REGION Network 65: [Ax] Movimento PTRK da Pos1 Ribalta + Tempo Assestamento ==a==> Pos2 Ribalta
   RUNG wire#powerrail
      "PTrk_Presence"(Item := "PTrk".A0301.P["PTRK_A0301_Ribalta_Pos1"])
      "PTrk_Absence"(Item := "PTrk".A0301.P["PTRK_A0301_Ribalta_Pos2"])
      I_Contact( #Ctrl.TRK.Ribaltatore.MoveToPos1 )
      Contact( #CIn.Ribaltatore.Solleva_Rib.Work )
      Contact( #CIn.Ribaltatore.Sts_Ribaltatore.Pos1_Reached )
      { S7_Templates := "time_type := Time" } #TON.Delay_Pos1Ribalta.TON(pt := "PPrf_MAIN".ON_WORK.A0301_A0302.Ribaltatore.Pos_1_Delay, et =>)
      Contact( #TON.Delay_Pos1Ribalta.Q )
      wire#w1
      I_Contact( #CIn.Ribaltatore.Sts_Ribaltatore.Pos2_Reached )
      wire#w2
      Coil( #Ctrl.TRK.Ribaltatore.MoveToPos2 )
   END_RUNG
   RUNG wire#powerrail
      "PTrk_Presence"(Item := "PTrk".A0301.P["PTRK_A0301_Ribalta_Pos2"])
      I_Contact( #Ctrl.TRK.Ribaltatore.MoveToPos1 )
      I_Contact( #Ctrl.TRK.Ribaltatore.MoveToPos3 )
   END_RUNG wire#w1
   RUNG wire#powerrail
      Contact( #Ctrl.TRK.Ribaltatore.MoveToPos2 )
      I_Contact( #CIn.Ribaltatore.Sts_Ribaltatore.Pos2_Reached )
   END_RUNG wire#w2
   RUNG wire#powerrail
      I_Contact( #Ctrl.TRK.Ribaltatore.MoveToPos2 )
      Contact( #CIn.Ribaltatore.Sts_Ribaltatore.Pos2_Reached )
      "PTrk_Presence"(Item := "PTrk".A0301.P["PTRK_A0301_Ribalta_Pos1"])
      "PTrk_Absence"(Item := "PTrk".A0301.P["PTRK_A0301_Ribalta_Pos2"])
      Move(in := "PTrk".A0301.P["PTRK_A0301_Ribalta_Pos1"], out1 => "PTrk".A0301.P["PTRK_A0301_Ribalta_Pos2"])
      "PTrk_Presence"(Item := "PTrk".A0301.P["PTRK_A0301_Ribalta_Pos2"])
      Move(in := "PTrk".Empty, out1 => "PTrk".A0301.P["PTRK_A0301_Ribalta_Pos1"])
   END_RUNG
   // the same network as SCL:
   "PTrk_Presence"(Item := "PTrk".A0301.P["PTRK_A0301_Ribalta_Pos1"], ENO => #_w1);
   "PTrk_Absence"(EN := #_w1, Item := "PTrk".A0301.P["PTRK_A0301_Ribalta_Pos2"], ENO => #_w2);
   #TON.Delay_Pos1Ribalta.TON(IN := #_w2 AND NOT #Ctrl.TRK.Ribaltatore.MoveToPos1 AND #CIn.Ribaltatore.Solleva_Rib.Work AND #CIn.Ribaltatore.Sts_Ribaltatore.Pos1_Reached,
                           PT := "PPrf_MAIN".ON_WORK.A0301_A0302.Ribaltatore.Pos_1_Delay);
   "PTrk_Presence"(Item := "PTrk".A0301.P["PTRK_A0301_Ribalta_Pos2"], ENO => #_w3);
   #Ctrl.TRK.Ribaltatore.MoveToPos2 := (((#TON.Delay_Pos1Ribalta.Q AND #TON.Delay_Pos1Ribalta.Q) OR (#_w3 AND NOT #Ctrl.TRK.Ribaltatore.MoveToPos1 AND NOT #Ctrl.TRK.Ribaltatore.MoveToPos3)) AND NOT #CIn.Ribaltatore.Sts_Ribaltatore.Pos2_Reached) OR (#Ctrl.TRK.Ribaltatore.MoveToPos2 AND NOT #CIn.Ribaltatore.Sts_Ribaltatore.Pos2_Reached);
   "PTrk_Presence"(EN := NOT #Ctrl.TRK.Ribaltatore.MoveToPos2 AND #CIn.Ribaltatore.Sts_Ribaltatore.Pos2_Reached,
                   Item := "PTrk".A0301.P["PTRK_A0301_Ribalta_Pos1"],
                   ENO => #_w4);
   "PTrk_Absence"(EN := #_w4, Item := "PTrk".A0301.P["PTRK_A0301_Ribalta_Pos2"], ENO => #_w5);
   IF #_w5 THEN
       "PTrk".A0301.P["PTRK_A0301_Ribalta_Pos2"] := "PTrk".A0301.P["PTRK_A0301_Ribalta_Pos1"];
   END_IF;
   "PTrk_Presence"(EN := #_w5, Item := "PTrk".A0301.P["PTRK_A0301_Ribalta_Pos2"], ENO => #_w6);
   IF #_w6 THEN "PTrk".A0301.P["PTRK_A0301_Ribalta_Pos1"] := "PTrk".Empty; END_IF;
END_REGION

REGION Network 66: [Ax] Movimento PTRK da Pos2 Ribalta ==a==> Pos3 Ribalta
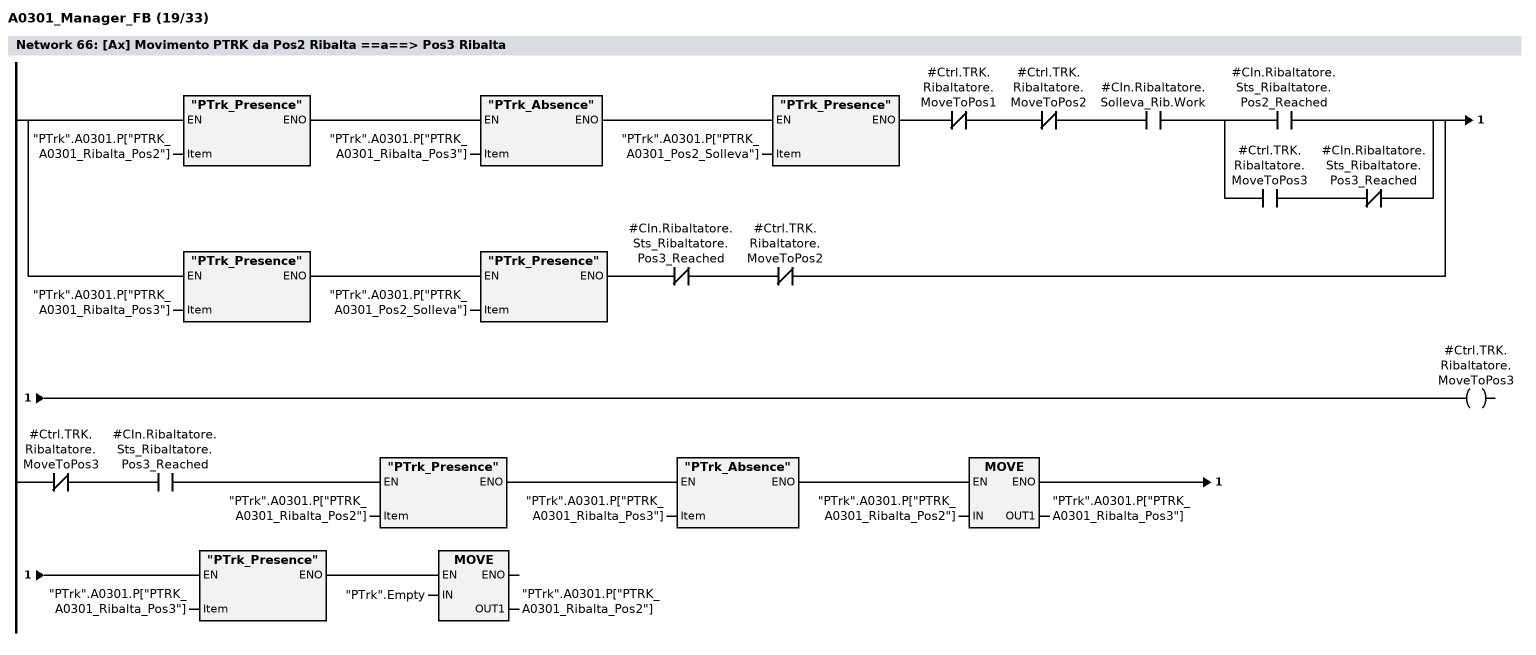
   RUNG wire#powerrail
      "PTrk_Presence"(Item := "PTrk".A0301.P["PTRK_A0301_Ribalta_Pos2"])
      "PTrk_Absence"(Item := "PTrk".A0301.P["PTRK_A0301_Ribalta_Pos3"])
      "PTrk_Presence"(Item := "PTrk".A0301.P["PTRK_A0301_Pos2_Solleva"])
      I_Contact( #Ctrl.TRK.Ribaltatore.MoveToPos1 )
      I_Contact( #Ctrl.TRK.Ribaltatore.MoveToPos2 )
      Contact( #CIn.Ribaltatore.Solleva_Rib.Work )
      wire#w1
      Contact( #CIn.Ribaltatore.Sts_Ribaltatore.Pos2_Reached )
      wire#w2
      Coil( #Ctrl.TRK.Ribaltatore.MoveToPos3 )
   END_RUNG
   RUNG wire#w1
      Contact( #Ctrl.TRK.Ribaltatore.MoveToPos3 )
      I_Contact( #CIn.Ribaltatore.Sts_Ribaltatore.Pos3_Reached )
   END_RUNG wire#w2
   RUNG wire#powerrail
      "PTrk_Presence"(Item := "PTrk".A0301.P["PTRK_A0301_Ribalta_Pos3"])
      "PTrk_Presence"(Item := "PTrk".A0301.P["PTRK_A0301_Pos2_Solleva"])
      I_Contact( #CIn.Ribaltatore.Sts_Ribaltatore.Pos3_Reached )
      I_Contact( #Ctrl.TRK.Ribaltatore.MoveToPos2 )
   END_RUNG wire#w2
   RUNG wire#powerrail
      I_Contact( #Ctrl.TRK.Ribaltatore.MoveToPos3 )
      Contact( #CIn.Ribaltatore.Sts_Ribaltatore.Pos3_Reached )
      "PTrk_Presence"(Item := "PTrk".A0301.P["PTRK_A0301_Ribalta_Pos2"])
      "PTrk_Absence"(Item := "PTrk".A0301.P["PTRK_A0301_Ribalta_Pos3"])
      Move(in := "PTrk".A0301.P["PTRK_A0301_Ribalta_Pos2"], out1 => "PTrk".A0301.P["PTRK_A0301_Ribalta_Pos3"])
      "PTrk_Presence"(Item := "PTrk".A0301.P["PTRK_A0301_Ribalta_Pos3"])
      Move(in := "PTrk".Empty, out1 => "PTrk".A0301.P["PTRK_A0301_Ribalta_Pos2"])
   END_RUNG
   // the same network as SCL:
   "PTrk_Presence"(Item := "PTrk".A0301.P["PTRK_A0301_Ribalta_Pos2"], ENO => #_w1);
   "PTrk_Absence"(EN := #_w1, Item := "PTrk".A0301.P["PTRK_A0301_Ribalta_Pos3"], ENO => #_w2);
   "PTrk_Presence"(EN := #_w2, Item := "PTrk".A0301.P["PTRK_A0301_Pos2_Solleva"], ENO => #_w3);
   "PTrk_Presence"(Item := "PTrk".A0301.P["PTRK_A0301_Ribalta_Pos3"], ENO => #_w4);
   "PTrk_Presence"(EN := #_w4, Item := "PTrk".A0301.P["PTRK_A0301_Pos2_Solleva"], ENO => #_w5);
   #Ctrl.TRK.Ribaltatore.MoveToPos3 := (#_w3 AND NOT #Ctrl.TRK.Ribaltatore.MoveToPos1 AND NOT #Ctrl.TRK.Ribaltatore.MoveToPos2 AND #CIn.Ribaltatore.Solleva_Rib.Work AND (#CIn.Ribaltatore.Sts_Ribaltatore.Pos2_Reached OR (#Ctrl.TRK.Ribaltatore.MoveToPos3 AND NOT #CIn.Ribaltatore.Sts_Ribaltatore.Pos3_Reached))) OR (#_w5 AND NOT #CIn.Ribaltatore.Sts_Ribaltatore.Pos3_Reached AND NOT #Ctrl.TRK.Ribaltatore.MoveToPos2);
   "PTrk_Presence"(EN := NOT #Ctrl.TRK.Ribaltatore.MoveToPos3 AND #CIn.Ribaltatore.Sts_Ribaltatore.Pos3_Reached,
                   Item := "PTrk".A0301.P["PTRK_A0301_Ribalta_Pos2"],
                   ENO => #_w6);
   "PTrk_Absence"(EN := #_w6, Item := "PTrk".A0301.P["PTRK_A0301_Ribalta_Pos3"], ENO => #_w7);
   IF #_w7 THEN
       "PTrk".A0301.P["PTRK_A0301_Ribalta_Pos3"] := "PTrk".A0301.P["PTRK_A0301_Ribalta_Pos2"];
   END_IF;
   "PTrk_Presence"(EN := #_w7, Item := "PTrk".A0301.P["PTRK_A0301_Ribalta_Pos3"], ENO => #_w8);
   IF #_w8 THEN "PTrk".A0301.P["PTRK_A0301_Ribalta_Pos2"] := "PTrk".Empty; END_IF;
END_REGION

REGION Network 67: <+>
END_REGION

REGION Network 68: << GESTIONE MOVIMENTO RIBALTATORE / SOLLEVA RIBALTATORE >>
END_REGION

REGION Network 69: [Ax] Ribaltatore - COut Manager
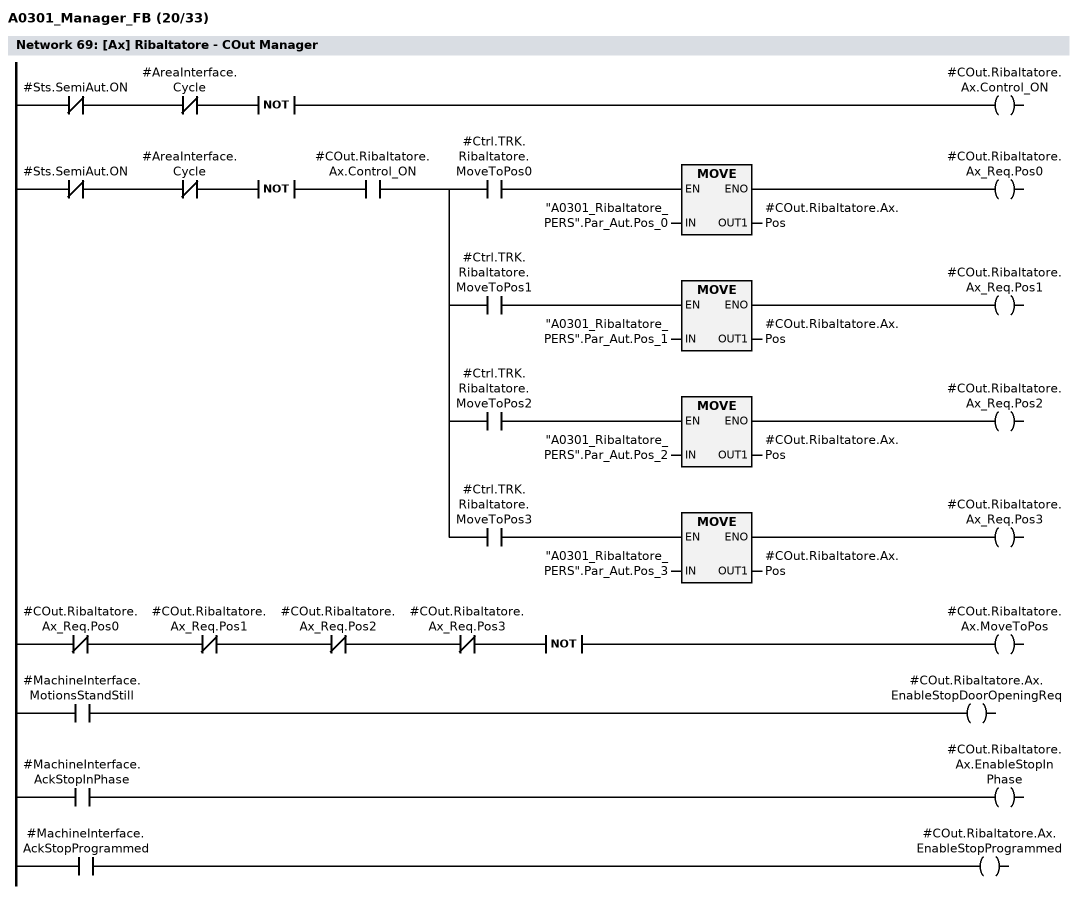
   RUNG wire#powerrail
      I_Contact( #Sts.SemiAut.ON )
      I_Contact( #AreaInterface.Cycle )
      Not()
      Coil( #COut.Ribaltatore.Ax.Control_ON )
   END_RUNG
   RUNG wire#powerrail
      I_Contact( #Sts.SemiAut.ON )
      I_Contact( #AreaInterface.Cycle )
      Not()
      Contact( #COut.Ribaltatore.Ax.Control_ON )
      wire#w1
      Contact( #Ctrl.TRK.Ribaltatore.MoveToPos0 )
      Move(in := "A0301_Ribaltatore_PERS".Par_Aut.Pos_0, out1 => #COut.Ribaltatore.Ax.Pos)
      Coil( #COut.Ribaltatore.Ax_Req.Pos0 )
   END_RUNG
   RUNG wire#w1
      Contact( #Ctrl.TRK.Ribaltatore.MoveToPos1 )
      Move(in := "A0301_Ribaltatore_PERS".Par_Aut.Pos_1, out1 => #COut.Ribaltatore.Ax.Pos)
      Coil( #COut.Ribaltatore.Ax_Req.Pos1 )
   END_RUNG
   RUNG wire#w1
      Contact( #Ctrl.TRK.Ribaltatore.MoveToPos2 )
      Move(in := "A0301_Ribaltatore_PERS".Par_Aut.Pos_2, out1 => #COut.Ribaltatore.Ax.Pos)
      Coil( #COut.Ribaltatore.Ax_Req.Pos2 )
   END_RUNG
   RUNG wire#w1
      Contact( #Ctrl.TRK.Ribaltatore.MoveToPos3 )
      Move(in := "A0301_Ribaltatore_PERS".Par_Aut.Pos_3, out1 => #COut.Ribaltatore.Ax.Pos)
      Coil( #COut.Ribaltatore.Ax_Req.Pos3 )
   END_RUNG
   RUNG wire#powerrail
      I_Contact( #COut.Ribaltatore.Ax_Req.Pos0 )
      I_Contact( #COut.Ribaltatore.Ax_Req.Pos1 )
      I_Contact( #COut.Ribaltatore.Ax_Req.Pos2 )
      I_Contact( #COut.Ribaltatore.Ax_Req.Pos3 )
      Not()
      Coil( #COut.Ribaltatore.Ax.MoveToPos )
   END_RUNG
   RUNG wire#powerrail
      Contact( #MachineInterface.MotionsStandStill )
      Coil( #COut.Ribaltatore.Ax.EnableStopDoorOpeningReq )
   END_RUNG
   RUNG wire#powerrail
      Contact( #MachineInterface.AckStopInPhase )
      Coil( #COut.Ribaltatore.Ax.EnableStopInPhase )
   END_RUNG
   RUNG wire#powerrail
      Contact( #MachineInterface.AckStopProgrammed )
      Coil( #COut.Ribaltatore.Ax.EnableStopProgrammed )
   END_RUNG
   // the same network as SCL:
   #COut.Ribaltatore.Ax.Control_ON := NOT (NOT #Sts.SemiAut.ON AND NOT #AreaInterface.Cycle);
   #_w1 := NOT (NOT #Sts.SemiAut.ON AND NOT #AreaInterface.Cycle) AND #COut.Ribaltatore.Ax.Control_ON;
   #_w2 := #_w1 AND #Ctrl.TRK.Ribaltatore.MoveToPos0;
   IF #_w2 THEN #COut.Ribaltatore.Ax.Pos := "A0301_Ribaltatore_PERS".Par_Aut.Pos_0; END_IF;
   #COut.Ribaltatore.Ax_Req.Pos0 := #_w2;
   #_w3 := #_w1 AND #Ctrl.TRK.Ribaltatore.MoveToPos1;
   IF #_w3 THEN #COut.Ribaltatore.Ax.Pos := "A0301_Ribaltatore_PERS".Par_Aut.Pos_1; END_IF;
   #COut.Ribaltatore.Ax_Req.Pos1 := #_w3;
   #_w4 := #_w1 AND #Ctrl.TRK.Ribaltatore.MoveToPos2;
   IF #_w4 THEN #COut.Ribaltatore.Ax.Pos := "A0301_Ribaltatore_PERS".Par_Aut.Pos_2; END_IF;
   #COut.Ribaltatore.Ax_Req.Pos2 := #_w4;
   #_w5 := #_w1 AND #Ctrl.TRK.Ribaltatore.MoveToPos3;
   IF #_w5 THEN #COut.Ribaltatore.Ax.Pos := "A0301_Ribaltatore_PERS".Par_Aut.Pos_3; END_IF;
   #COut.Ribaltatore.Ax_Req.Pos3 := #_w5;
   #COut.Ribaltatore.Ax.MoveToPos := NOT (NOT #COut.Ribaltatore.Ax_Req.Pos0 AND NOT #COut.Ribaltatore.Ax_Req.Pos1 AND NOT #COut.Ribaltatore.Ax_Req.Pos2 AND NOT #COut.Ribaltatore.Ax_Req.Pos3);
   #COut.Ribaltatore.Ax.EnableStopDoorOpeningReq := #MachineInterface.MotionsStandStill;
   #COut.Ribaltatore.Ax.EnableStopInPhase := #MachineInterface.AckStopInPhase;
   #COut.Ribaltatore.Ax.EnableStopProgrammed := #MachineInterface.AckStopProgrammed;
END_REGION

REGION Network 70: [Ax] Ribaltatore - RIFERIMENTI Velocità
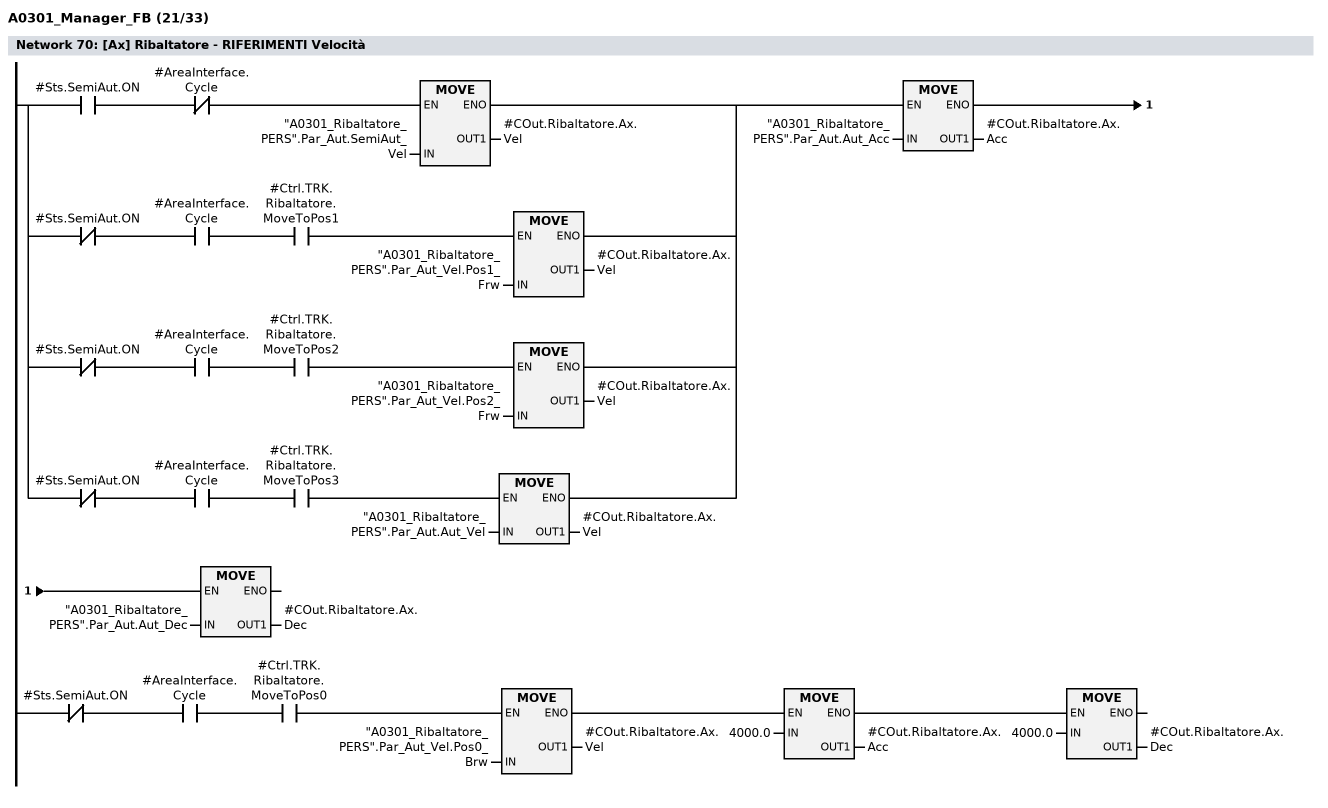
   RUNG wire#powerrail
      Contact( #Sts.SemiAut.ON )
      I_Contact( #AreaInterface.Cycle )
      Move(in := "A0301_Ribaltatore_PERS".Par_Aut.SemiAut_Vel, out1 => #COut.Ribaltatore.Ax.Vel)
      wire#w1
      Move(in := "A0301_Ribaltatore_PERS".Par_Aut.Aut_Acc, out1 => #COut.Ribaltatore.Ax.Acc)
      Move(in := "A0301_Ribaltatore_PERS".Par_Aut.Aut_Dec, out1 => #COut.Ribaltatore.Ax.Dec)
   END_RUNG
   RUNG wire#powerrail
      I_Contact( #Sts.SemiAut.ON )
      Contact( #AreaInterface.Cycle )
      Contact( #Ctrl.TRK.Ribaltatore.MoveToPos1 )
      Move(in := "A0301_Ribaltatore_PERS".Par_Aut_Vel.Pos1_Frw, out1 => #COut.Ribaltatore.Ax.Vel)
   END_RUNG wire#w1
   RUNG wire#powerrail
      I_Contact( #Sts.SemiAut.ON )
      Contact( #AreaInterface.Cycle )
      Contact( #Ctrl.TRK.Ribaltatore.MoveToPos2 )
      Move(in := "A0301_Ribaltatore_PERS".Par_Aut_Vel.Pos2_Frw, out1 => #COut.Ribaltatore.Ax.Vel)
   END_RUNG wire#w1
   RUNG wire#powerrail
      I_Contact( #Sts.SemiAut.ON )
      Contact( #AreaInterface.Cycle )
      Contact( #Ctrl.TRK.Ribaltatore.MoveToPos3 )
      Move(in := "A0301_Ribaltatore_PERS".Par_Aut.Aut_Vel, out1 => #COut.Ribaltatore.Ax.Vel)
   END_RUNG wire#w1
   RUNG wire#powerrail
      I_Contact( #Sts.SemiAut.ON )
      Contact( #AreaInterface.Cycle )
      Contact( #Ctrl.TRK.Ribaltatore.MoveToPos0 )
      Move(in := "A0301_Ribaltatore_PERS".Par_Aut_Vel.Pos0_Brw, out1 => #COut.Ribaltatore.Ax.Vel)
      Move(in := 4000.0, out1 => #COut.Ribaltatore.Ax.Acc)
      Move(in := 4000.0, out1 => #COut.Ribaltatore.Ax.Dec)
   END_RUNG
   // the same network as SCL:
   #_w1 := #Sts.SemiAut.ON AND NOT #AreaInterface.Cycle;
   IF #_w1 THEN #COut.Ribaltatore.Ax.Vel := "A0301_Ribaltatore_PERS".Par_Aut.SemiAut_Vel; END_IF;
   #_w2 := NOT #Sts.SemiAut.ON AND #AreaInterface.Cycle AND #Ctrl.TRK.Ribaltatore.MoveToPos1;
   IF #_w2 THEN #COut.Ribaltatore.Ax.Vel := "A0301_Ribaltatore_PERS".Par_Aut_Vel.Pos1_Frw; END_IF;
   #_w3 := NOT #Sts.SemiAut.ON AND #AreaInterface.Cycle AND #Ctrl.TRK.Ribaltatore.MoveToPos2;
   IF #_w3 THEN #COut.Ribaltatore.Ax.Vel := "A0301_Ribaltatore_PERS".Par_Aut_Vel.Pos2_Frw; END_IF;
   #_w4 := NOT #Sts.SemiAut.ON AND #AreaInterface.Cycle AND #Ctrl.TRK.Ribaltatore.MoveToPos3;
   IF #_w4 THEN #COut.Ribaltatore.Ax.Vel := "A0301_Ribaltatore_PERS".Par_Aut.Aut_Vel; END_IF;
   IF #_w1 OR #_w2 OR #_w3 OR #_w4 THEN
       #COut.Ribaltatore.Ax.Acc := "A0301_Ribaltatore_PERS".Par_Aut.Aut_Acc;
       #COut.Ribaltatore.Ax.Dec := "A0301_Ribaltatore_PERS".Par_Aut.Aut_Dec;
   END_IF;
   IF NOT #Sts.SemiAut.ON AND #AreaInterface.Cycle AND #Ctrl.TRK.Ribaltatore.MoveToPos0 THEN
       #COut.Ribaltatore.Ax.Vel := "A0301_Ribaltatore_PERS".Par_Aut_Vel.Pos0_Brw;
       #COut.Ribaltatore.Ax.Acc := 4000.0;
       #COut.Ribaltatore.Ax.Dec := 4000.0;
   END_IF;
END_REGION

REGION Network 71: P [Solleva] Ribaltatore - COut Manager
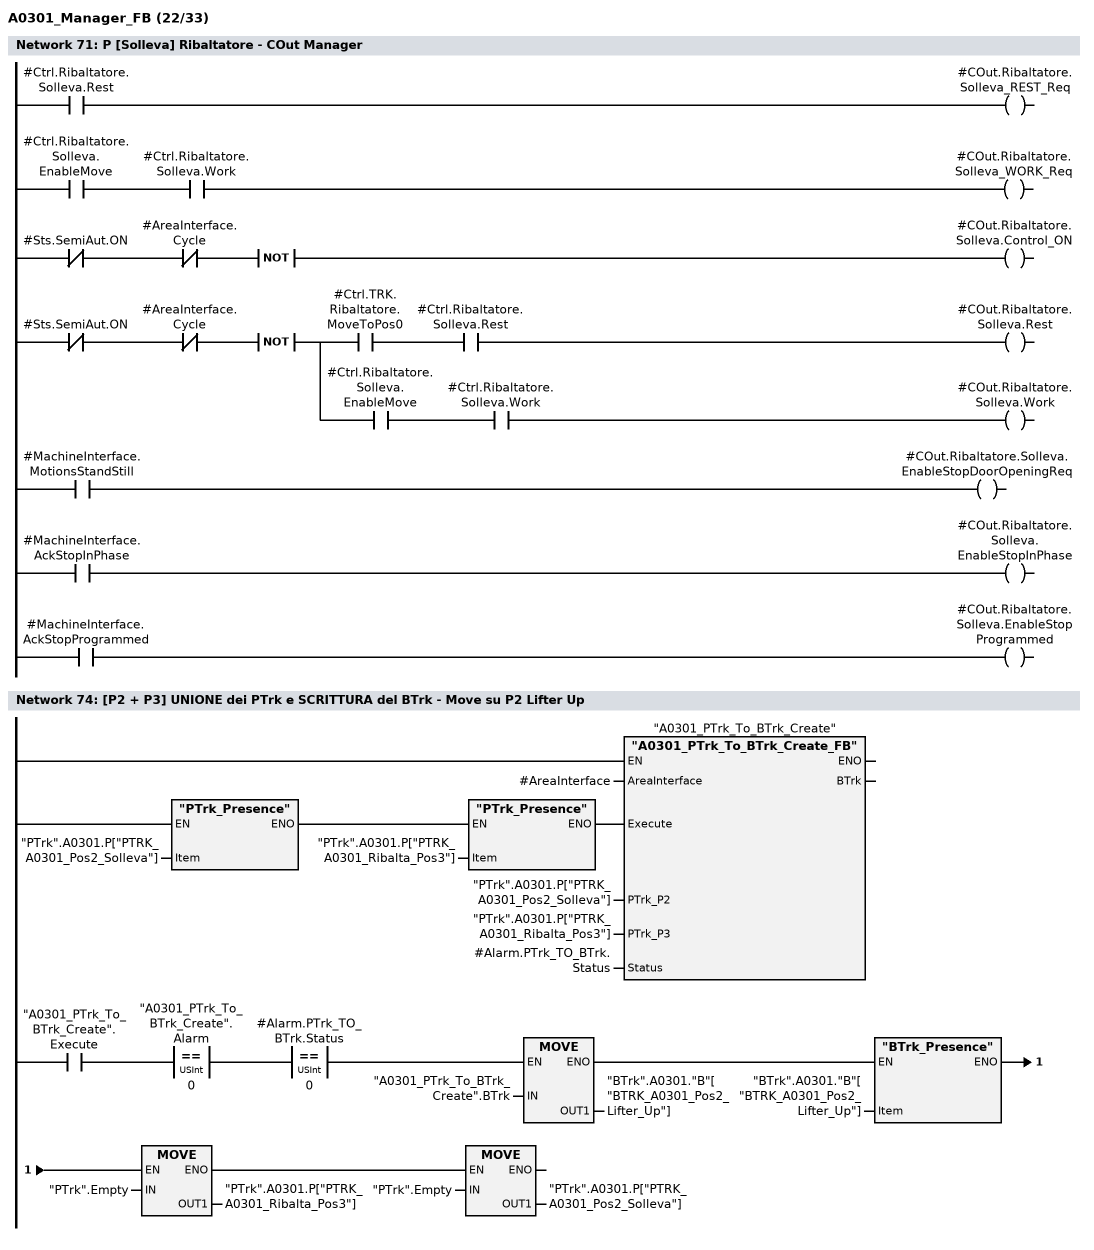
   RUNG wire#powerrail
      Contact( #Ctrl.Ribaltatore.Solleva.Rest )
      Coil( #COut.Ribaltatore.Solleva_REST_Req )
   END_RUNG
   RUNG wire#powerrail
      Contact( #Ctrl.Ribaltatore.Solleva.EnableMove )
      Contact( #Ctrl.Ribaltatore.Solleva.Work )
      Coil( #COut.Ribaltatore.Solleva_WORK_Req )
   END_RUNG
   RUNG wire#powerrail
      I_Contact( #Sts.SemiAut.ON )
      I_Contact( #AreaInterface.Cycle )
      Not()
      Coil( #COut.Ribaltatore.Solleva.Control_ON )
   END_RUNG
   RUNG wire#powerrail
      I_Contact( #Sts.SemiAut.ON )
      I_Contact( #AreaInterface.Cycle )
      Not()
      wire#w1
      Contact( #Ctrl.TRK.Ribaltatore.MoveToPos0 )
      Contact( #Ctrl.Ribaltatore.Solleva.Rest )
      Coil( #COut.Ribaltatore.Solleva.Rest )
   END_RUNG
   RUNG wire#w1
      Contact( #Ctrl.Ribaltatore.Solleva.EnableMove )
      Contact( #Ctrl.Ribaltatore.Solleva.Work )
      Coil( #COut.Ribaltatore.Solleva.Work )
   END_RUNG
   RUNG wire#powerrail
      Contact( #MachineInterface.MotionsStandStill )
      Coil( #COut.Ribaltatore.Solleva.EnableStopDoorOpeningReq )
   END_RUNG
   RUNG wire#powerrail
      Contact( #MachineInterface.AckStopInPhase )
      Coil( #COut.Ribaltatore.Solleva.EnableStopInPhase )
   END_RUNG
   RUNG wire#powerrail
      Contact( #MachineInterface.AckStopProgrammed )
      Coil( #COut.Ribaltatore.Solleva.EnableStopProgrammed )
   END_RUNG
   // the same network as SCL:
   #COut.Ribaltatore.Solleva_REST_Req := #Ctrl.Ribaltatore.Solleva.Rest;
   #COut.Ribaltatore.Solleva_WORK_Req := #Ctrl.Ribaltatore.Solleva.EnableMove AND #Ctrl.Ribaltatore.Solleva.Work;
   #COut.Ribaltatore.Solleva.Control_ON := NOT (NOT #Sts.SemiAut.ON AND NOT #AreaInterface.Cycle);
   #_w1 := NOT (NOT #Sts.SemiAut.ON AND NOT #AreaInterface.Cycle);
   #COut.Ribaltatore.Solleva.Rest := #_w1 AND #Ctrl.TRK.Ribaltatore.MoveToPos0 AND #Ctrl.Ribaltatore.Solleva.Rest;
   #COut.Ribaltatore.Solleva.Work := #_w1 AND #Ctrl.Ribaltatore.Solleva.EnableMove AND #Ctrl.Ribaltatore.Solleva.Work;
   #COut.Ribaltatore.Solleva.EnableStopDoorOpeningReq := #MachineInterface.MotionsStandStill;
   #COut.Ribaltatore.Solleva.EnableStopInPhase := #MachineInterface.AckStopInPhase;
   #COut.Ribaltatore.Solleva.EnableStopProgrammed := #MachineInterface.AckStopProgrammed;
END_REGION

REGION Network 73: <<<<<<<<<<<<<<<<<<< CREAZIONE TRAKING BTRK >>>>>>>>>>>>>>>>>>>>>
END_REGION

REGION Network 74: [P2 + P3] UNIONE dei PTrk e SCRITTURA del BTrk - Move su P2 Lifter Up
   RUNG wire#powerrail
      "A0301_PTrk_To_BTrk_Create"(Execute := wire#w1, AreaInterface := #AreaInterface, PTrk_P2 := "PTrk".A0301.P["PTRK_A0301_Pos2_Solleva"], PTrk_P3 := "PTrk".A0301.P["PTRK_A0301_Ribalta_Pos3"], Status := #Alarm.PTrk_TO_BTrk.Status, BTrk =>)
   END_RUNG
   RUNG wire#powerrail
      "PTrk_Presence"(Item := "PTrk".A0301.P["PTRK_A0301_Pos2_Solleva"])
      "PTrk_Presence"(Item := "PTrk".A0301.P["PTRK_A0301_Ribalta_Pos3"])
   END_RUNG wire#w1
   RUNG wire#powerrail
      Contact( "A0301_PTrk_To_BTrk_Create".Execute )
      { S7_Templates := "SrcType := USInt" } EQ_Contact(in1 := "A0301_PTrk_To_BTrk_Create".Alarm, in2 := 0)
      { S7_Templates := "SrcType := USInt" } EQ_Contact(in1 := #Alarm.PTrk_TO_BTrk.Status, in2 := 0)
      Move(in := "A0301_PTrk_To_BTrk_Create".BTrk, out1 => "BTrk".A0301."B"["BTRK_A0301_Pos2_Lifter_Up"])
      "BTrk_Presence"(Item := "BTrk".A0301."B"["BTRK_A0301_Pos2_Lifter_Up"])
      Move(in := "PTrk".Empty, out1 => "PTrk".A0301.P["PTRK_A0301_Ribalta_Pos3"])
      Move(in := "PTrk".Empty, out1 => "PTrk".A0301.P["PTRK_A0301_Pos2_Solleva"])
   END_RUNG
   // the same network as SCL:
   "PTrk_Presence"(Item := "PTrk".A0301.P["PTRK_A0301_Pos2_Solleva"], ENO => #_w1);
   "PTrk_Presence"(EN := #_w1, Item := "PTrk".A0301.P["PTRK_A0301_Ribalta_Pos3"], ENO => #_w2);
   "A0301_PTrk_To_BTrk_Create"(AreaInterface := #AreaInterface,   // "A0301_PTrk_To_BTrk_Create_FB"
                           Execute := #_w2,
                           PTrk_P2 := "PTrk".A0301.P["PTRK_A0301_Pos2_Solleva"],
                           PTrk_P3 := "PTrk".A0301.P["PTRK_A0301_Ribalta_Pos3"],
                           Status := #Alarm.PTrk_TO_BTrk.Status);
   IF "A0301_PTrk_To_BTrk_Create".Execute AND ("A0301_PTrk_To_BTrk_Create".Alarm = 0) AND (#Alarm.PTrk_TO_BTrk.Status = 0) THEN
       "BTrk".A0301."B"["BTRK_A0301_Pos2_Lifter_Up"] := "A0301_PTrk_To_BTrk_Create".BTrk;
   END_IF;
   "BTrk_Presence"(EN := "A0301_PTrk_To_BTrk_Create".Execute AND ("A0301_PTrk_To_BTrk_Create".Alarm = 0) AND (#Alarm.PTrk_TO_BTrk.Status = 0),
                   Item := "BTrk".A0301."B"["BTRK_A0301_Pos2_Lifter_Up"],
                   ENO => #_w3);
   IF #_w3 THEN
       "PTrk".A0301.P["PTRK_A0301_Ribalta_Pos3"] := "PTrk".Empty;
       "PTrk".A0301.P["PTRK_A0301_Pos2_Solleva"] := "PTrk".Empty;
   END_IF;
END_REGION

REGION Network 76: <<<<<<<<<<< POSIZIONE 4 >>>>>>>>>>>
END_REGION

REGION Network 77 (SCL): [P4] Reset allarmi
   IF #AreaInterface.RstAlarms THEN
       #Alarm.P2toP4_NotReached := FALSE;
   END_IF;
END_REGION

REGION Network 78: [P4] Movimento BTRK da Pos2 Up ==a==> Pos2 Down
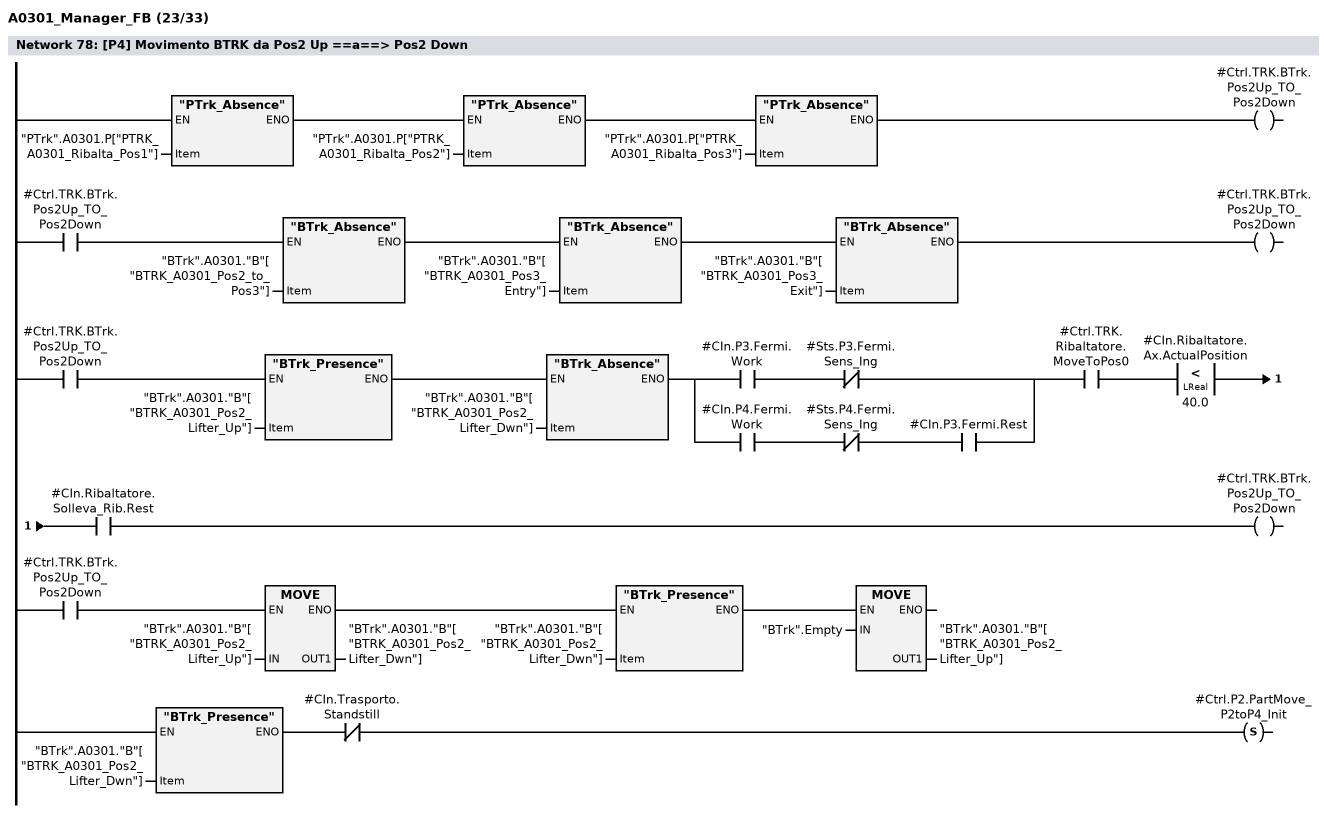
   RUNG wire#powerrail
      "PTrk_Absence"(Item := "PTrk".A0301.P["PTRK_A0301_Ribalta_Pos1"])
      "PTrk_Absence"(Item := "PTrk".A0301.P["PTRK_A0301_Ribalta_Pos2"])
      "PTrk_Absence"(Item := "PTrk".A0301.P["PTRK_A0301_Ribalta_Pos3"])
      Coil( #Ctrl.TRK.BTrk.Pos2Up_TO_Pos2Down )
   END_RUNG
   RUNG wire#powerrail
      Contact( #Ctrl.TRK.BTrk.Pos2Up_TO_Pos2Down )
      "BTrk_Absence"(Item := "BTrk".A0301."B"["BTRK_A0301_Pos2_to_Pos3"])
      "BTrk_Absence"(Item := "BTrk".A0301."B"["BTRK_A0301_Pos3_Entry"])
      "BTrk_Absence"(Item := "BTrk".A0301."B"["BTRK_A0301_Pos3_Exit"])
      Coil( #Ctrl.TRK.BTrk.Pos2Up_TO_Pos2Down )
   END_RUNG
   RUNG wire#powerrail
      Contact( #Ctrl.TRK.BTrk.Pos2Up_TO_Pos2Down )
      "BTrk_Presence"(Item := "BTrk".A0301."B"["BTRK_A0301_Pos2_Lifter_Up"])
      "BTrk_Absence"(Item := "BTrk".A0301."B"["BTRK_A0301_Pos2_Lifter_Dwn"])
      wire#w1
      Contact( #CIn.P3.Fermi.Work )
      I_Contact( #Sts.P3.Fermi.Sens_Ing )
      wire#w2
      Contact( #Ctrl.TRK.Ribaltatore.MoveToPos0 )
      { S7_Templates := "SrcType := LReal" } LT_Contact(in1 := #CIn.Ribaltatore.Ax.ActualPosition, in2 := 40.0)
      Contact( #CIn.Ribaltatore.Solleva_Rib.Rest )
      Coil( #Ctrl.TRK.BTrk.Pos2Up_TO_Pos2Down )
   END_RUNG
   RUNG wire#w1
      Contact( #CIn.P4.Fermi.Work )
      I_Contact( #Sts.P4.Fermi.Sens_Ing )
      Contact( #CIn.P3.Fermi.Rest )
   END_RUNG wire#w2
   RUNG wire#powerrail
      Contact( #Ctrl.TRK.BTrk.Pos2Up_TO_Pos2Down )
      Move(in := "BTrk".A0301."B"["BTRK_A0301_Pos2_Lifter_Up"], out1 => "BTrk".A0301."B"["BTRK_A0301_Pos2_Lifter_Dwn"])
      "BTrk_Presence"(Item := "BTrk".A0301."B"["BTRK_A0301_Pos2_Lifter_Dwn"])
      Move(in := "BTrk".Empty, out1 => "BTrk".A0301."B"["BTRK_A0301_Pos2_Lifter_Up"])
   END_RUNG
   RUNG wire#powerrail
      "BTrk_Presence"(Item := "BTrk".A0301."B"["BTRK_A0301_Pos2_Lifter_Dwn"])
      I_Contact( #CIn.Trasporto.Standstill )
      S_Coil( #Ctrl.P2.PartMove_P2toP4_Init )
   END_RUNG
   // the same network as SCL:
   "PTrk_Absence"(Item := "PTrk".A0301.P["PTRK_A0301_Ribalta_Pos1"], ENO => #_w1);
   "PTrk_Absence"(EN := #_w1, Item := "PTrk".A0301.P["PTRK_A0301_Ribalta_Pos2"], ENO => #_w2);
   "PTrk_Absence"(EN := #_w2, Item := "PTrk".A0301.P["PTRK_A0301_Ribalta_Pos3"], ENO => #_w3);
   #Ctrl.TRK.BTrk.Pos2Up_TO_Pos2Down := #_w3;
   "BTrk_Absence"(EN := #Ctrl.TRK.BTrk.Pos2Up_TO_Pos2Down,
                  Item := "BTrk".A0301."B"["BTRK_A0301_Pos2_to_Pos3"],
                  ENO => #_w4);
   "BTrk_Absence"(EN := #_w4, Item := "BTrk".A0301."B"["BTRK_A0301_Pos3_Entry"], ENO => #_w5);
   "BTrk_Absence"(EN := #_w5, Item := "BTrk".A0301."B"["BTRK_A0301_Pos3_Exit"], ENO => #_w6);
   #Ctrl.TRK.BTrk.Pos2Up_TO_Pos2Down := #_w6;
   "BTrk_Presence"(EN := #Ctrl.TRK.BTrk.Pos2Up_TO_Pos2Down,
                   Item := "BTrk".A0301."B"["BTRK_A0301_Pos2_Lifter_Up"],
                   ENO => #_w7);
   "BTrk_Absence"(EN := #_w7, Item := "BTrk".A0301."B"["BTRK_A0301_Pos2_Lifter_Dwn"], ENO => #_w8);
   #Ctrl.TRK.BTrk.Pos2Up_TO_Pos2Down := #_w8 AND ((#CIn.P3.Fermi.Work AND NOT #Sts.P3.Fermi.Sens_Ing) OR (#CIn.P4.Fermi.Work AND NOT #Sts.P4.Fermi.Sens_Ing AND #CIn.P3.Fermi.Rest)) AND #Ctrl.TRK.Ribaltatore.MoveToPos0 AND (#CIn.Ribaltatore.Ax.ActualPosition < 40.0) AND #CIn.Ribaltatore.Solleva_Rib.Rest;
   IF #Ctrl.TRK.BTrk.Pos2Up_TO_Pos2Down THEN
       "BTrk".A0301."B"["BTRK_A0301_Pos2_Lifter_Dwn"] := "BTrk".A0301."B"["BTRK_A0301_Pos2_Lifter_Up"];
   END_IF;
   "BTrk_Presence"(EN := #Ctrl.TRK.BTrk.Pos2Up_TO_Pos2Down,
                   Item := "BTrk".A0301."B"["BTRK_A0301_Pos2_Lifter_Dwn"],
                   ENO => #_w9);
   IF #_w9 THEN "BTrk".A0301."B"["BTRK_A0301_Pos2_Lifter_Up"] := "BTrk".Empty; END_IF;
   "BTrk_Presence"(Item := "BTrk".A0301."B"["BTRK_A0301_Pos2_Lifter_Dwn"], ENO => #_w10);
   IF #_w10 AND NOT #CIn.Trasporto.Standstill THEN #Ctrl.P2.PartMove_P2toP4_Init := TRUE; END_IF;
END_REGION

REGION Network 79: == Monitoraggio spazio di trasporto del movimento BTrk da Pos.2 Down a Pos.4 Entry ==
   // Controllo la posizione salvata da Pos.2 Lifter Down + Distanza sensori Pos.2 / Pos.4 = Target da raggiungere
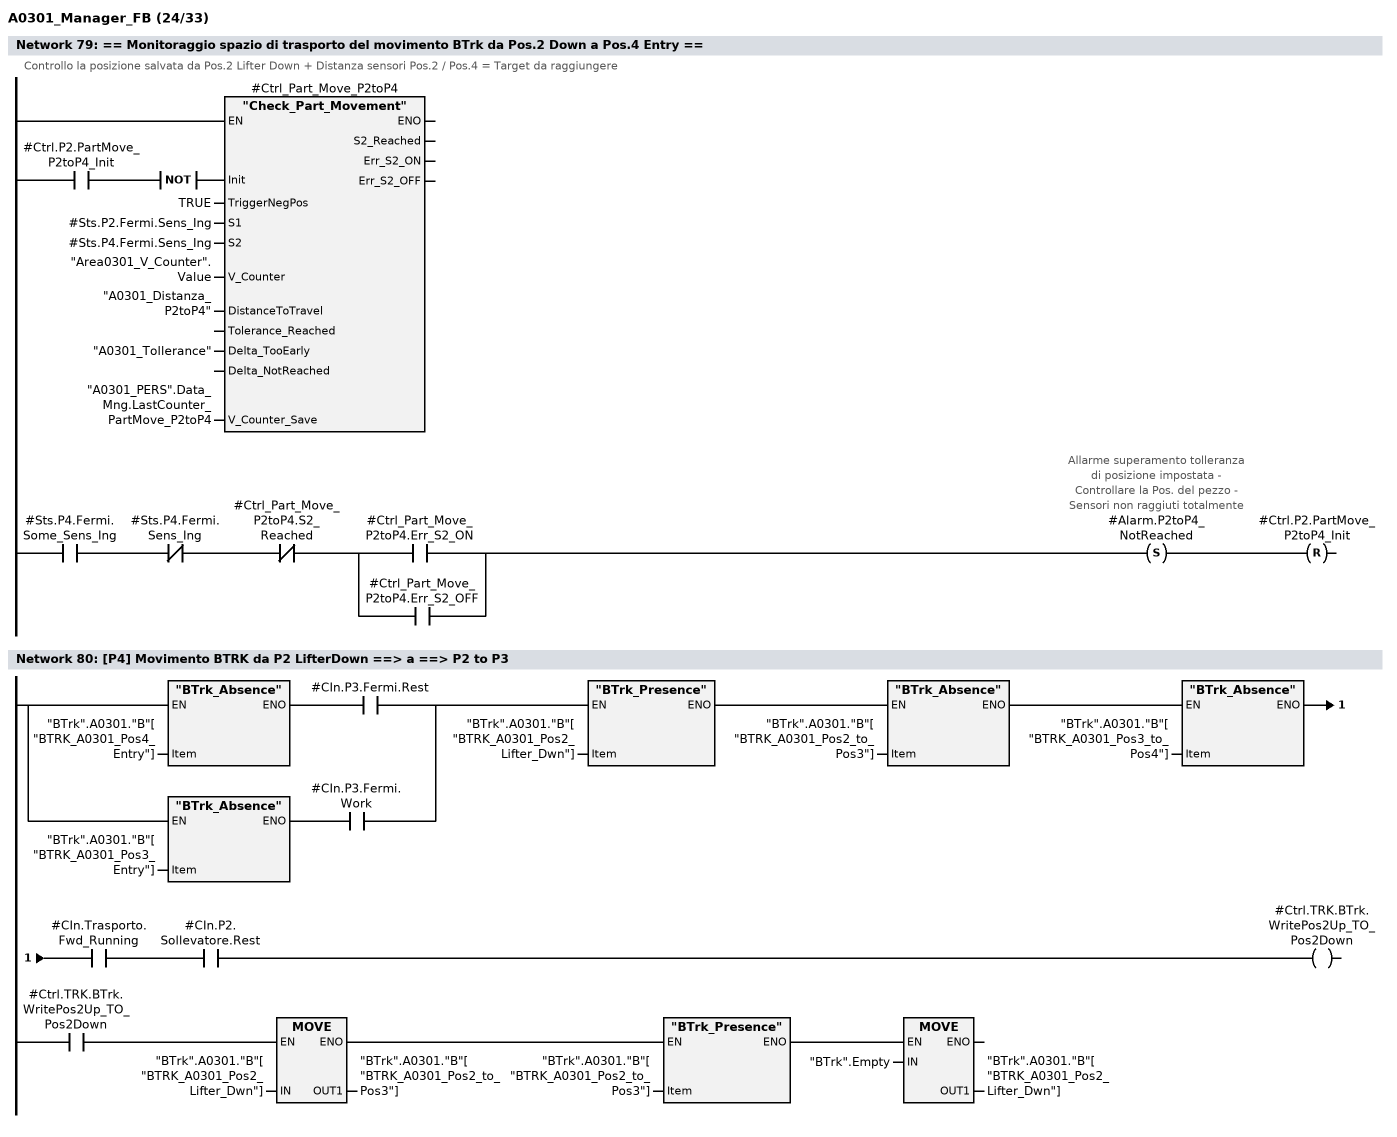
   RUNG wire#powerrail
      #Ctrl_Part_Move_P2toP4(Init := wire#w1, TriggerNegPos := TRUE, S1 := #Sts.P2.Fermi.Sens_Ing, S2 := #Sts.P4.Fermi.Sens_Ing, V_Counter := "Area0301_V_Counter".Value, DistanceToTravel := "A0301_Distanza_P2toP4", Tolerance_Reached :=, Delta_TooEarly := "A0301_Tollerance", Delta_NotReached :=, V_Counter_Save := "A0301_PERS".Data_Mng.LastCounter_PartMove_P2toP4, S2_Reached =>, Err_S2_ON =>, Err_S2_OFF =>)
   END_RUNG
   RUNG wire#powerrail
      Contact( #Ctrl.P2.PartMove_P2toP4_Init )
      Not()
   END_RUNG wire#w1
   RUNG wire#powerrail
      Contact( #Sts.P4.Fermi.Some_Sens_Ing )
      I_Contact( #Sts.P4.Fermi.Sens_Ing )
      I_Contact( #Ctrl_Part_Move_P2toP4.S2_Reached )
      wire#w2
      Contact( #Ctrl_Part_Move_P2toP4.Err_S2_ON )
      wire#w3
      S_Coil( #Alarm.P2toP4_NotReached )   // Allarme superamento tolleranza di posizione impostata - Controllare la Pos. del pezzo - Sensori non raggiuti totalmente
      R_Coil( #Ctrl.P2.PartMove_P2toP4_Init )
   END_RUNG
   RUNG wire#w2
      Contact( #Ctrl_Part_Move_P2toP4.Err_S2_OFF )
   END_RUNG wire#w3
   // the same network as SCL:
   #Ctrl_Part_Move_P2toP4(Init := NOT #Ctrl.P2.PartMove_P2toP4_Init,   // "Check_Part_Movement"
                          TriggerNegPos := TRUE,
                          S1 := #Sts.P2.Fermi.Sens_Ing,
                          S2 := #Sts.P4.Fermi.Sens_Ing,
                          V_Counter := "Area0301_V_Counter".Value,
                          DistanceToTravel := "A0301_Distanza_P2toP4",
                          Delta_TooEarly := "A0301_Tollerance",
                          V_Counter_Save := "A0301_PERS".Data_Mng.LastCounter_PartMove_P2toP4);
   IF #Sts.P4.Fermi.Some_Sens_Ing AND NOT #Sts.P4.Fermi.Sens_Ing AND NOT #Ctrl_Part_Move_P2toP4.S2_Reached AND (#Ctrl_Part_Move_P2toP4.Err_S2_ON OR #Ctrl_Part_Move_P2toP4.Err_S2_OFF) THEN
       #Alarm.P2toP4_NotReached := TRUE;   // Allarme superamento tolleranza di posizione impostata - Controllare la Pos. del pezzo - Sensori non raggiuti totalmente
       #Ctrl.P2.PartMove_P2toP4_Init := FALSE;
   END_IF;
END_REGION

REGION Network 80: [P4] Movimento BTRK da P2 LifterDown ==> a ==> P2 to P3
   RUNG wire#powerrail
      "BTrk_Absence"(Item := "BTrk".A0301."B"["BTRK_A0301_Pos4_Entry"])
      Contact( #CIn.P3.Fermi.Rest )
      wire#w1
      "BTrk_Presence"(Item := "BTrk".A0301."B"["BTRK_A0301_Pos2_Lifter_Dwn"])
      "BTrk_Absence"(Item := "BTrk".A0301."B"["BTRK_A0301_Pos2_to_Pos3"])
      "BTrk_Absence"(Item := "BTrk".A0301."B"["BTRK_A0301_Pos3_to_Pos4"])
      Contact( #CIn.Trasporto.Fwd_Running )
      Contact( #CIn.P2.Sollevatore.Rest )
      Coil( #Ctrl.TRK.BTrk.WritePos2Up_TO_Pos2Down )
   END_RUNG
   RUNG wire#powerrail
      "BTrk_Absence"(Item := "BTrk".A0301."B"["BTRK_A0301_Pos3_Entry"])
      Contact( #CIn.P3.Fermi.Work )
   END_RUNG wire#w1
   RUNG wire#powerrail
      Contact( #Ctrl.TRK.BTrk.WritePos2Up_TO_Pos2Down )
      Move(in := "BTrk".A0301."B"["BTRK_A0301_Pos2_Lifter_Dwn"], out1 => "BTrk".A0301."B"["BTRK_A0301_Pos2_to_Pos3"])
      "BTrk_Presence"(Item := "BTrk".A0301."B"["BTRK_A0301_Pos2_to_Pos3"])
      Move(in := "BTrk".Empty, out1 => "BTrk".A0301."B"["BTRK_A0301_Pos2_Lifter_Dwn"])
   END_RUNG
   // the same network as SCL:
   "BTrk_Absence"(Item := "BTrk".A0301."B"["BTRK_A0301_Pos4_Entry"], ENO => #_w1);
   "BTrk_Absence"(Item := "BTrk".A0301."B"["BTRK_A0301_Pos3_Entry"], ENO => #_w2);
   "BTrk_Presence"(EN := (#_w1 AND #CIn.P3.Fermi.Rest) OR (#_w2 AND #CIn.P3.Fermi.Work),
                   Item := "BTrk".A0301."B"["BTRK_A0301_Pos2_Lifter_Dwn"],
                   ENO => #_w3);
   "BTrk_Absence"(EN := #_w3, Item := "BTrk".A0301."B"["BTRK_A0301_Pos2_to_Pos3"], ENO => #_w4);
   "BTrk_Absence"(EN := #_w4, Item := "BTrk".A0301."B"["BTRK_A0301_Pos3_to_Pos4"], ENO => #_w5);
   #Ctrl.TRK.BTrk.WritePos2Up_TO_Pos2Down := #_w5 AND #CIn.Trasporto.Fwd_Running AND #CIn.P2.Sollevatore.Rest;
   IF #Ctrl.TRK.BTrk.WritePos2Up_TO_Pos2Down THEN
       "BTrk".A0301."B"["BTRK_A0301_Pos2_to_Pos3"] := "BTrk".A0301."B"["BTRK_A0301_Pos2_Lifter_Dwn"];
   END_IF;
   "BTrk_Presence"(EN := #Ctrl.TRK.BTrk.WritePos2Up_TO_Pos2Down,
                   Item := "BTrk".A0301."B"["BTRK_A0301_Pos2_to_Pos3"],
                   ENO => #_w6);
   IF #_w6 THEN "BTrk".A0301."B"["BTRK_A0301_Pos2_Lifter_Dwn"] := "BTrk".Empty; END_IF;
END_REGION

REGION Network 81: [P4] Movimento BTRK da P2 To Pos3==> a ==> P3 Entry
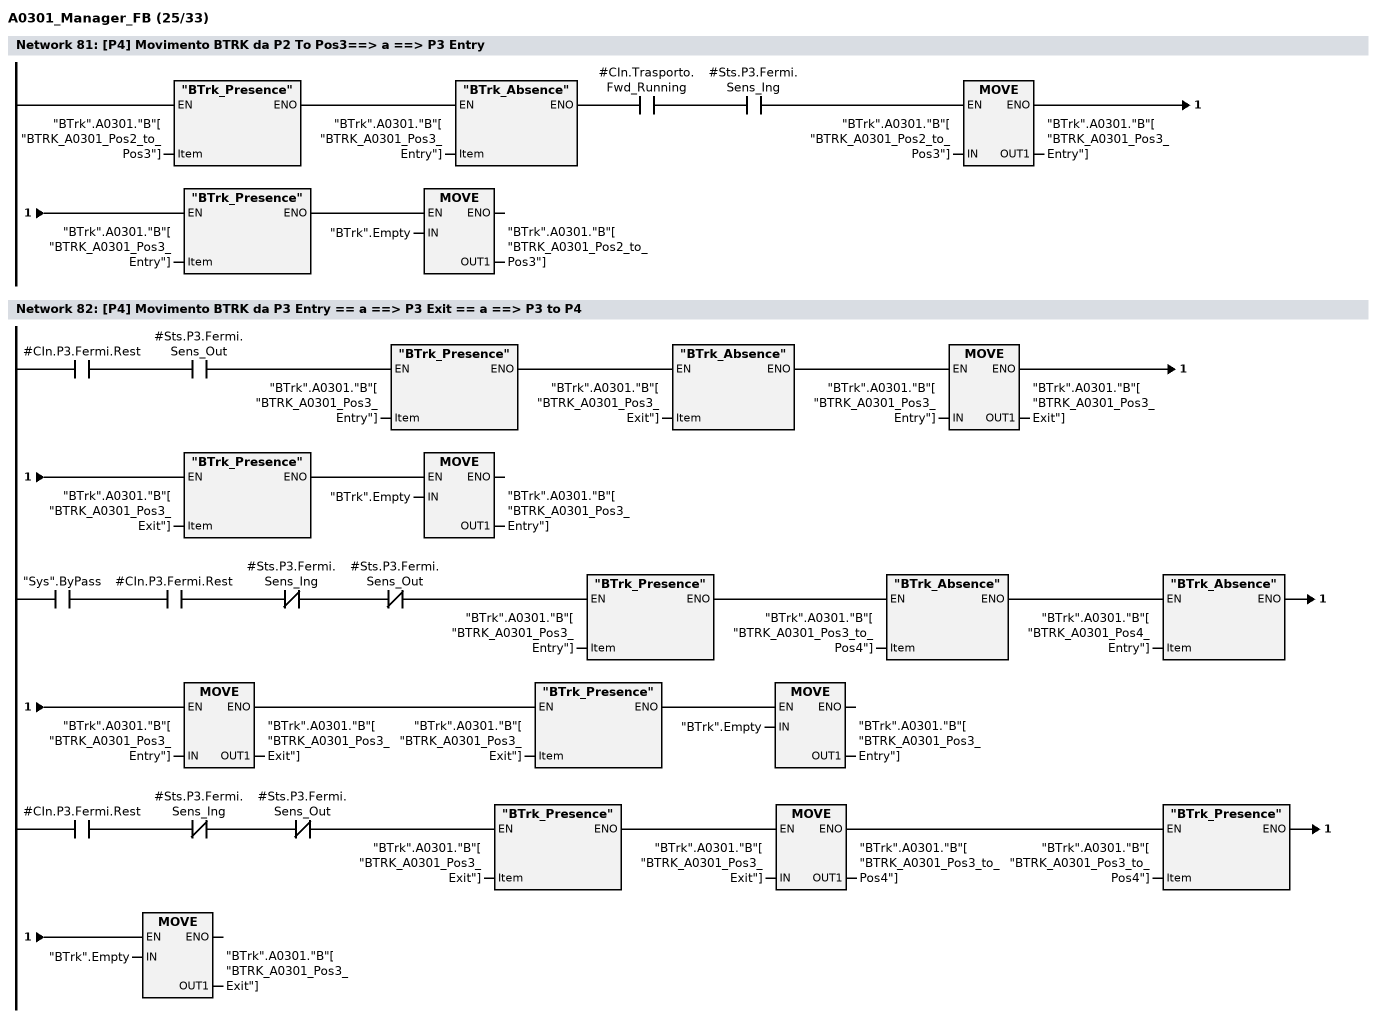
   RUNG wire#powerrail
      "BTrk_Presence"(Item := "BTrk".A0301."B"["BTRK_A0301_Pos2_to_Pos3"])
      "BTrk_Absence"(Item := "BTrk".A0301."B"["BTRK_A0301_Pos3_Entry"])
      Contact( #CIn.Trasporto.Fwd_Running )
      Contact( #Sts.P3.Fermi.Sens_Ing )
      Move(in := "BTrk".A0301."B"["BTRK_A0301_Pos2_to_Pos3"], out1 => "BTrk".A0301."B"["BTRK_A0301_Pos3_Entry"])
      "BTrk_Presence"(Item := "BTrk".A0301."B"["BTRK_A0301_Pos3_Entry"])
      Move(in := "BTrk".Empty, out1 => "BTrk".A0301."B"["BTRK_A0301_Pos2_to_Pos3"])
   END_RUNG
   // the same network as SCL:
   "BTrk_Presence"(Item := "BTrk".A0301."B"["BTRK_A0301_Pos2_to_Pos3"], ENO => #_w1);
   "BTrk_Absence"(EN := #_w1, Item := "BTrk".A0301."B"["BTRK_A0301_Pos3_Entry"], ENO => #_w2);
   IF #_w2 AND #CIn.Trasporto.Fwd_Running AND #Sts.P3.Fermi.Sens_Ing THEN
       "BTrk".A0301."B"["BTRK_A0301_Pos3_Entry"] := "BTrk".A0301."B"["BTRK_A0301_Pos2_to_Pos3"];
   END_IF;
   "BTrk_Presence"(EN := #_w2 AND #CIn.Trasporto.Fwd_Running AND #Sts.P3.Fermi.Sens_Ing,
                   Item := "BTrk".A0301."B"["BTRK_A0301_Pos3_Entry"],
                   ENO => #_w3);
   IF #_w3 THEN "BTrk".A0301."B"["BTRK_A0301_Pos2_to_Pos3"] := "BTrk".Empty; END_IF;
END_REGION

REGION Network 82: [P4] Movimento BTRK da P3 Entry == a ==> P3 Exit == a ==> P3 to P4
   RUNG wire#powerrail
      Contact( #CIn.P3.Fermi.Rest )
      Contact( #Sts.P3.Fermi.Sens_Out )
      "BTrk_Presence"(Item := "BTrk".A0301."B"["BTRK_A0301_Pos3_Entry"])
      "BTrk_Absence"(Item := "BTrk".A0301."B"["BTRK_A0301_Pos3_Exit"])
      Move(in := "BTrk".A0301."B"["BTRK_A0301_Pos3_Entry"], out1 => "BTrk".A0301."B"["BTRK_A0301_Pos3_Exit"])
      "BTrk_Presence"(Item := "BTrk".A0301."B"["BTRK_A0301_Pos3_Exit"])
      Move(in := "BTrk".Empty, out1 => "BTrk".A0301."B"["BTRK_A0301_Pos3_Entry"])
   END_RUNG
   RUNG wire#powerrail
      Contact( "Sys".ByPass )
      Contact( #CIn.P3.Fermi.Rest )
      I_Contact( #Sts.P3.Fermi.Sens_Ing )
      I_Contact( #Sts.P3.Fermi.Sens_Out )
      "BTrk_Presence"(Item := "BTrk".A0301."B"["BTRK_A0301_Pos3_Entry"])
      "BTrk_Absence"(Item := "BTrk".A0301."B"["BTRK_A0301_Pos3_to_Pos4"])
      "BTrk_Absence"(Item := "BTrk".A0301."B"["BTRK_A0301_Pos4_Entry"])
      Move(in := "BTrk".A0301."B"["BTRK_A0301_Pos3_Entry"], out1 => "BTrk".A0301."B"["BTRK_A0301_Pos3_Exit"])
      "BTrk_Presence"(Item := "BTrk".A0301."B"["BTRK_A0301_Pos3_Exit"])
      Move(in := "BTrk".Empty, out1 => "BTrk".A0301."B"["BTRK_A0301_Pos3_Entry"])
   END_RUNG
   RUNG wire#powerrail
      Contact( #CIn.P3.Fermi.Rest )
      I_Contact( #Sts.P3.Fermi.Sens_Ing )
      I_Contact( #Sts.P3.Fermi.Sens_Out )
      "BTrk_Presence"(Item := "BTrk".A0301."B"["BTRK_A0301_Pos3_Exit"])
      Move(in := "BTrk".A0301."B"["BTRK_A0301_Pos3_Exit"], out1 => "BTrk".A0301."B"["BTRK_A0301_Pos3_to_Pos4"])
      "BTrk_Presence"(Item := "BTrk".A0301."B"["BTRK_A0301_Pos3_to_Pos4"])
      Move(in := "BTrk".Empty, out1 => "BTrk".A0301."B"["BTRK_A0301_Pos3_Exit"])
   END_RUNG
   // the same network as SCL:
   "BTrk_Presence"(EN := #CIn.P3.Fermi.Rest AND #Sts.P3.Fermi.Sens_Out,
                   Item := "BTrk".A0301."B"["BTRK_A0301_Pos3_Entry"],
                   ENO => #_w1);
   "BTrk_Absence"(EN := #_w1, Item := "BTrk".A0301."B"["BTRK_A0301_Pos3_Exit"], ENO => #_w2);
   IF #_w2 THEN
       "BTrk".A0301."B"["BTRK_A0301_Pos3_Exit"] := "BTrk".A0301."B"["BTRK_A0301_Pos3_Entry"];
   END_IF;
   "BTrk_Presence"(EN := #_w2, Item := "BTrk".A0301."B"["BTRK_A0301_Pos3_Exit"], ENO => #_w3);
   IF #_w3 THEN "BTrk".A0301."B"["BTRK_A0301_Pos3_Entry"] := "BTrk".Empty; END_IF;
   "BTrk_Presence"(EN := "Sys".ByPass AND #CIn.P3.Fermi.Rest AND NOT #Sts.P3.Fermi.Sens_Ing AND NOT #Sts.P3.Fermi.Sens_Out,
                   Item := "BTrk".A0301."B"["BTRK_A0301_Pos3_Entry"],
                   ENO => #_w4);
   "BTrk_Absence"(EN := #_w4, Item := "BTrk".A0301."B"["BTRK_A0301_Pos3_to_Pos4"], ENO => #_w5);
   "BTrk_Absence"(EN := #_w5, Item := "BTrk".A0301."B"["BTRK_A0301_Pos4_Entry"], ENO => #_w6);
   IF #_w6 THEN
       "BTrk".A0301."B"["BTRK_A0301_Pos3_Exit"] := "BTrk".A0301."B"["BTRK_A0301_Pos3_Entry"];
   END_IF;
   "BTrk_Presence"(EN := #_w6, Item := "BTrk".A0301."B"["BTRK_A0301_Pos3_Exit"], ENO => #_w7);
   IF #_w7 THEN "BTrk".A0301."B"["BTRK_A0301_Pos3_Entry"] := "BTrk".Empty; END_IF;
   "BTrk_Presence"(EN := #CIn.P3.Fermi.Rest AND NOT #Sts.P3.Fermi.Sens_Ing AND NOT #Sts.P3.Fermi.Sens_Out,
                   Item := "BTrk".A0301."B"["BTRK_A0301_Pos3_Exit"],
                   ENO => #_w8);
   IF #_w8 THEN
       "BTrk".A0301."B"["BTRK_A0301_Pos3_to_Pos4"] := "BTrk".A0301."B"["BTRK_A0301_Pos3_Exit"];
   END_IF;
   "BTrk_Presence"(EN := #_w8, Item := "BTrk".A0301."B"["BTRK_A0301_Pos3_to_Pos4"], ENO => #_w9);
   IF #_w9 THEN "BTrk".A0301."B"["BTRK_A0301_Pos3_Exit"] := "BTrk".Empty; END_IF;
END_REGION

REGION Network 83: [P4] Movimento BTRK da P3 a P4 == a ==> P4 Entry
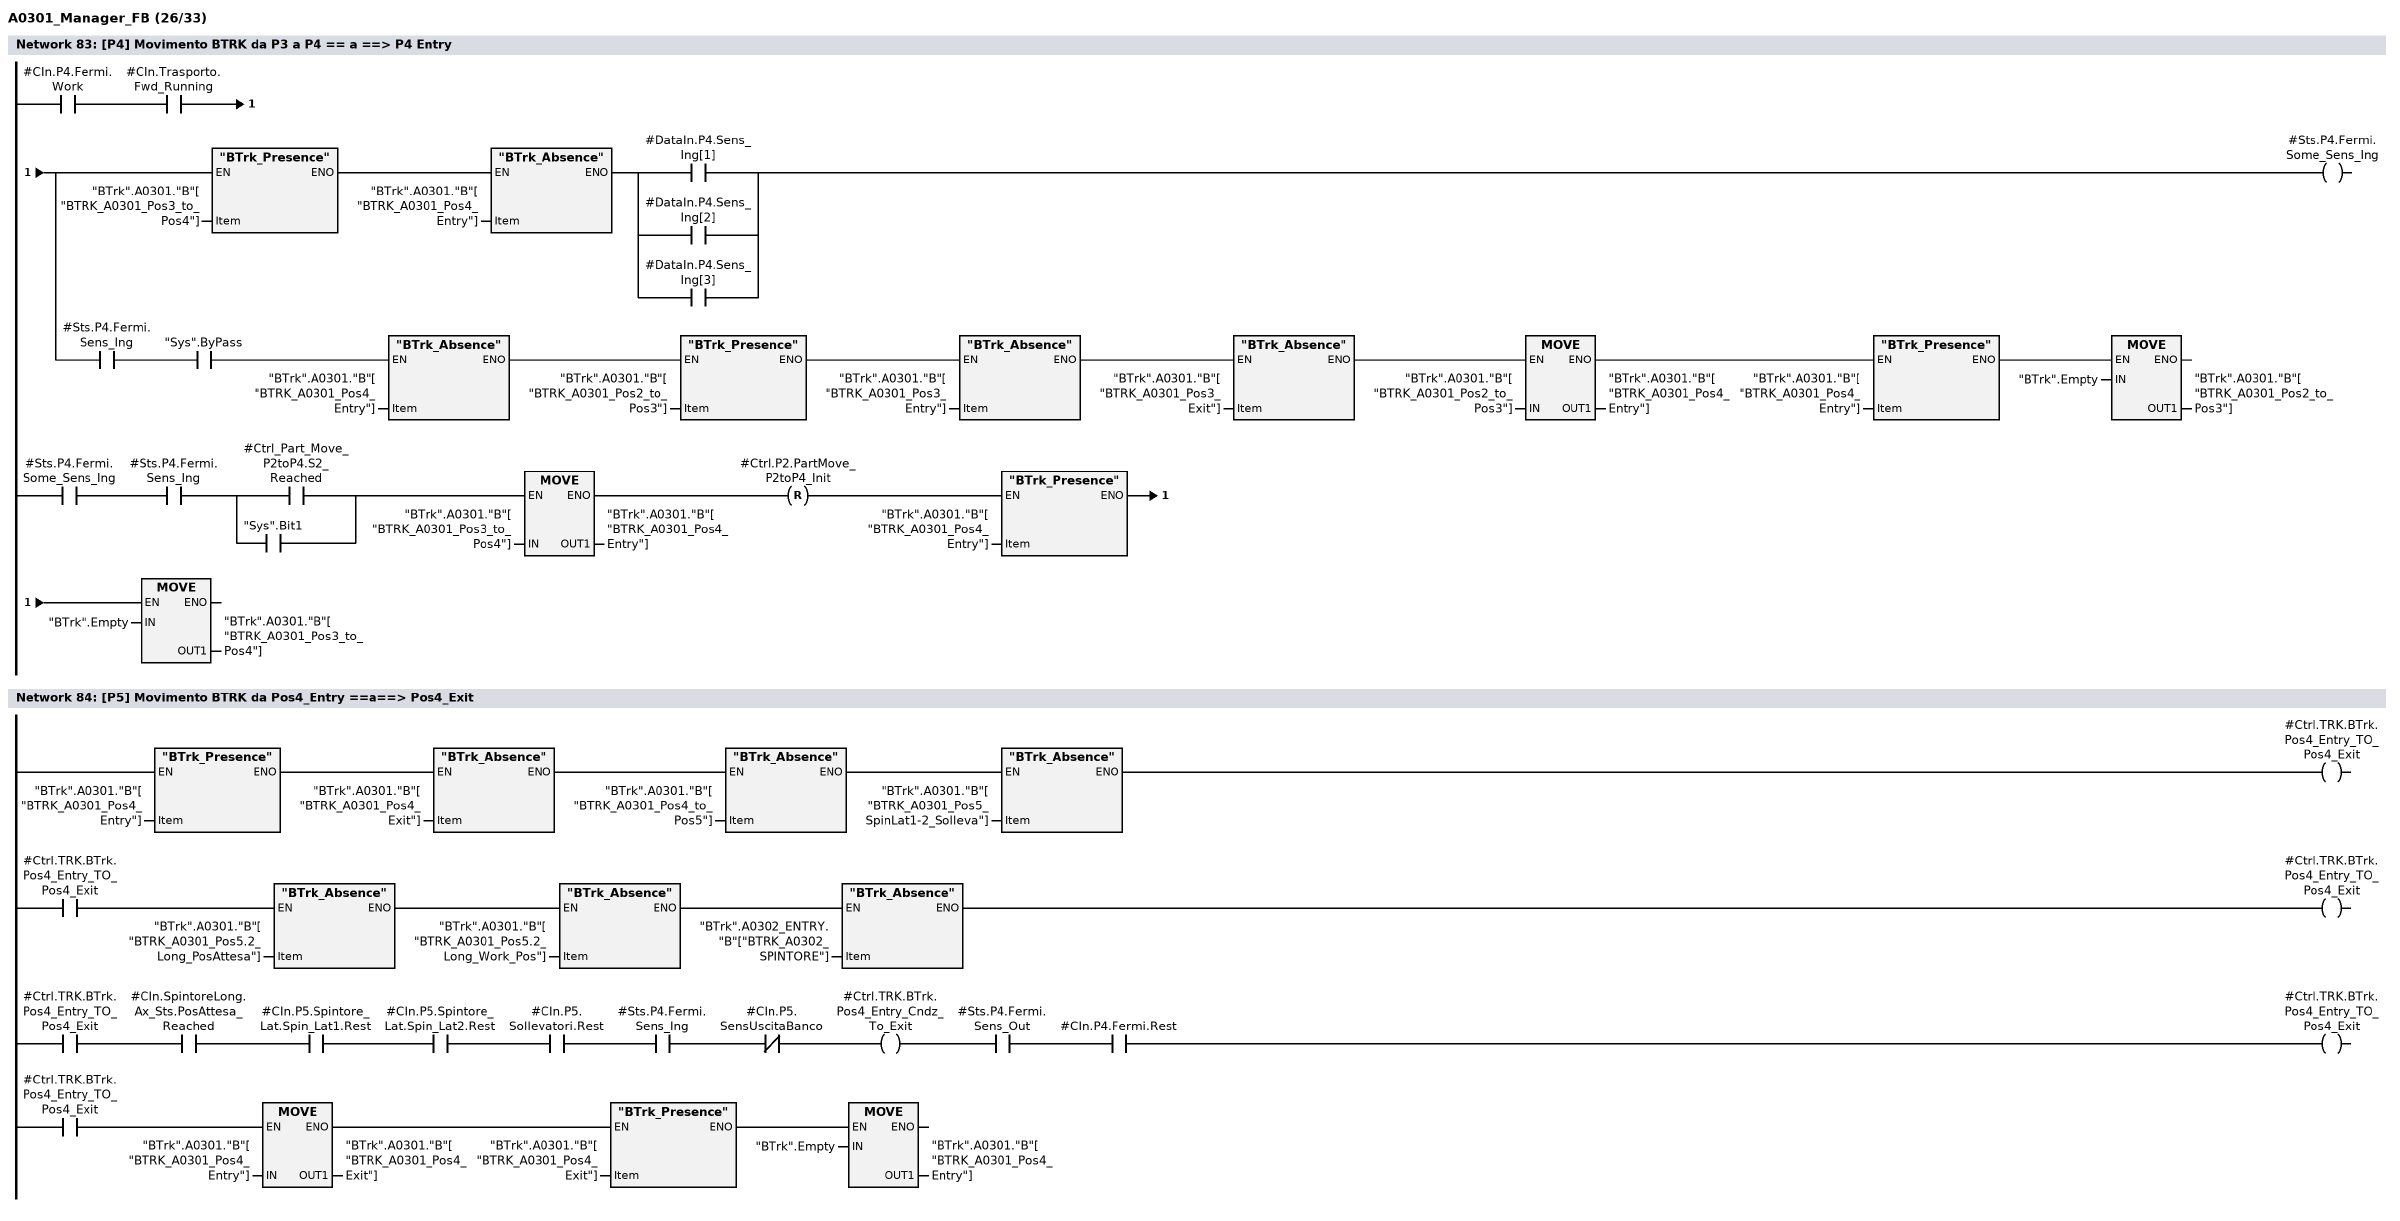
   RUNG wire#powerrail
      Contact( #CIn.P4.Fermi.Work )
      Contact( #CIn.Trasporto.Fwd_Running )
      wire#w1
      "BTrk_Presence"(Item := "BTrk".A0301."B"["BTRK_A0301_Pos3_to_Pos4"])
      "BTrk_Absence"(Item := "BTrk".A0301."B"["BTRK_A0301_Pos4_Entry"])
      wire#w2
      Contact( #DataIn.P4.Sens_Ing[1] )
      wire#w3
      Coil( #Sts.P4.Fermi.Some_Sens_Ing )
   END_RUNG
   RUNG wire#w2
      Contact( #DataIn.P4.Sens_Ing[2] )
   END_RUNG wire#w3
   RUNG wire#w2
      Contact( #DataIn.P4.Sens_Ing[3] )
   END_RUNG wire#w3
   RUNG wire#w1
      Contact( #Sts.P4.Fermi.Sens_Ing )
      Contact( "Sys".ByPass )
      "BTrk_Absence"(Item := "BTrk".A0301."B"["BTRK_A0301_Pos4_Entry"])
      "BTrk_Presence"(Item := "BTrk".A0301."B"["BTRK_A0301_Pos2_to_Pos3"])
      "BTrk_Absence"(Item := "BTrk".A0301."B"["BTRK_A0301_Pos3_Entry"])
      "BTrk_Absence"(Item := "BTrk".A0301."B"["BTRK_A0301_Pos3_Exit"])
      Move(in := "BTrk".A0301."B"["BTRK_A0301_Pos2_to_Pos3"], out1 => "BTrk".A0301."B"["BTRK_A0301_Pos4_Entry"])
      "BTrk_Presence"(Item := "BTrk".A0301."B"["BTRK_A0301_Pos4_Entry"])
      Move(in := "BTrk".Empty, out1 => "BTrk".A0301."B"["BTRK_A0301_Pos2_to_Pos3"])
   END_RUNG
   RUNG wire#powerrail
      Contact( #Sts.P4.Fermi.Some_Sens_Ing )
      Contact( #Sts.P4.Fermi.Sens_Ing )
      wire#w4
      Contact( #Ctrl_Part_Move_P2toP4.S2_Reached )
      wire#w5
      Move(in := "BTrk".A0301."B"["BTRK_A0301_Pos3_to_Pos4"], out1 => "BTrk".A0301."B"["BTRK_A0301_Pos4_Entry"])
      R_Coil( #Ctrl.P2.PartMove_P2toP4_Init )
      "BTrk_Presence"(Item := "BTrk".A0301."B"["BTRK_A0301_Pos4_Entry"])
      Move(in := "BTrk".Empty, out1 => "BTrk".A0301."B"["BTRK_A0301_Pos3_to_Pos4"])
   END_RUNG
   RUNG wire#w4
      Contact( "Sys".Bit1 )
   END_RUNG wire#w5
   // the same network as SCL:
   #_w1 := #CIn.P4.Fermi.Work AND #CIn.Trasporto.Fwd_Running;
   "BTrk_Presence"(EN := #_w1, Item := "BTrk".A0301."B"["BTRK_A0301_Pos3_to_Pos4"], ENO => #_w2);
   "BTrk_Absence"(EN := #_w2, Item := "BTrk".A0301."B"["BTRK_A0301_Pos4_Entry"], ENO => #_w3);
   #Sts.P4.Fermi.Some_Sens_Ing := #_w3 AND (#DataIn.P4.Sens_Ing[1] OR #DataIn.P4.Sens_Ing[2] OR #DataIn.P4.Sens_Ing[3]);
   "BTrk_Absence"(EN := #_w1 AND #Sts.P4.Fermi.Sens_Ing AND "Sys".ByPass,
                  Item := "BTrk".A0301."B"["BTRK_A0301_Pos4_Entry"],
                  ENO => #_w4);
   "BTrk_Presence"(EN := #_w4, Item := "BTrk".A0301."B"["BTRK_A0301_Pos2_to_Pos3"], ENO => #_w5);
   "BTrk_Absence"(EN := #_w5, Item := "BTrk".A0301."B"["BTRK_A0301_Pos3_Entry"], ENO => #_w6);
   "BTrk_Absence"(EN := #_w6, Item := "BTrk".A0301."B"["BTRK_A0301_Pos3_Exit"], ENO => #_w7);
   IF #_w7 THEN
       "BTrk".A0301."B"["BTRK_A0301_Pos4_Entry"] := "BTrk".A0301."B"["BTRK_A0301_Pos2_to_Pos3"];
   END_IF;
   "BTrk_Presence"(EN := #_w7, Item := "BTrk".A0301."B"["BTRK_A0301_Pos4_Entry"], ENO => #_w8);
   IF #_w8 THEN "BTrk".A0301."B"["BTRK_A0301_Pos2_to_Pos3"] := "BTrk".Empty; END_IF;
   IF #Sts.P4.Fermi.Some_Sens_Ing AND #Sts.P4.Fermi.Sens_Ing AND (#Ctrl_Part_Move_P2toP4.S2_Reached OR "Sys".Bit1) THEN
       "BTrk".A0301."B"["BTRK_A0301_Pos4_Entry"] := "BTrk".A0301."B"["BTRK_A0301_Pos3_to_Pos4"];
       #Ctrl.P2.PartMove_P2toP4_Init := FALSE;
   END_IF;
   "BTrk_Presence"(EN := #Sts.P4.Fermi.Some_Sens_Ing AND #Sts.P4.Fermi.Sens_Ing AND (#Ctrl_Part_Move_P2toP4.S2_Reached OR "Sys".Bit1),
                   Item := "BTrk".A0301."B"["BTRK_A0301_Pos4_Entry"],
                   ENO => #_w9);
   IF #_w9 THEN "BTrk".A0301."B"["BTRK_A0301_Pos3_to_Pos4"] := "BTrk".Empty; END_IF;
END_REGION

REGION Network 84: [P5] Movimento BTRK da Pos4_Entry ==a==> Pos4_Exit
   RUNG wire#powerrail
      "BTrk_Presence"(Item := "BTrk".A0301."B"["BTRK_A0301_Pos4_Entry"])
      "BTrk_Absence"(Item := "BTrk".A0301."B"["BTRK_A0301_Pos4_Exit"])
      "BTrk_Absence"(Item := "BTrk".A0301."B"["BTRK_A0301_Pos4_to_Pos5"])
      "BTrk_Absence"(Item := "BTrk".A0301."B"["BTRK_A0301_Pos5_SpinLat1-2_Solleva"])
      Coil( #Ctrl.TRK.BTrk.Pos4_Entry_TO_Pos4_Exit )
   END_RUNG
   RUNG wire#powerrail
      Contact( #Ctrl.TRK.BTrk.Pos4_Entry_TO_Pos4_Exit )
      "BTrk_Absence"(Item := "BTrk".A0301."B"["BTRK_A0301_Pos5.2_Long_PosAttesa"])
      "BTrk_Absence"(Item := "BTrk".A0301."B"["BTRK_A0301_Pos5.2_Long_Work_Pos"])
      "BTrk_Absence"(Item := "BTrk".A0302_ENTRY."B"["BTRK_A0302_SPINTORE"])
      Coil( #Ctrl.TRK.BTrk.Pos4_Entry_TO_Pos4_Exit )
   END_RUNG
   RUNG wire#powerrail
      Contact( #Ctrl.TRK.BTrk.Pos4_Entry_TO_Pos4_Exit )
      Contact( #CIn.SpintoreLong.Ax_Sts.PosAttesa_Reached )
      Contact( #CIn.P5.Spintore_Lat.Spin_Lat1.Rest )
      Contact( #CIn.P5.Spintore_Lat.Spin_Lat2.Rest )
      Contact( #CIn.P5.Sollevatori.Rest )
      Contact( #Sts.P4.Fermi.Sens_Ing )
      I_Contact( #CIn.P5.SensUscitaBanco )
      Coil( #Ctrl.TRK.BTrk.Pos4_Entry_Cndz_To_Exit )
      Contact( #Sts.P4.Fermi.Sens_Out )
      Contact( #CIn.P4.Fermi.Rest )
      Coil( #Ctrl.TRK.BTrk.Pos4_Entry_TO_Pos4_Exit )
   END_RUNG
   RUNG wire#powerrail
      Contact( #Ctrl.TRK.BTrk.Pos4_Entry_TO_Pos4_Exit )
      Move(in := "BTrk".A0301."B"["BTRK_A0301_Pos4_Entry"], out1 => "BTrk".A0301."B"["BTRK_A0301_Pos4_Exit"])
      "BTrk_Presence"(Item := "BTrk".A0301."B"["BTRK_A0301_Pos4_Exit"])
      Move(in := "BTrk".Empty, out1 => "BTrk".A0301."B"["BTRK_A0301_Pos4_Entry"])
   END_RUNG
   // the same network as SCL:
   "BTrk_Presence"(Item := "BTrk".A0301."B"["BTRK_A0301_Pos4_Entry"], ENO => #_w1);
   "BTrk_Absence"(EN := #_w1, Item := "BTrk".A0301."B"["BTRK_A0301_Pos4_Exit"], ENO => #_w2);
   "BTrk_Absence"(EN := #_w2, Item := "BTrk".A0301."B"["BTRK_A0301_Pos4_to_Pos5"], ENO => #_w3);
   "BTrk_Absence"(EN := #_w3, Item := "BTrk".A0301."B"["BTRK_A0301_Pos5_SpinLat1-2_Solleva"], ENO => #_w4);
   #Ctrl.TRK.BTrk.Pos4_Entry_TO_Pos4_Exit := #_w4;
   "BTrk_Absence"(EN := #Ctrl.TRK.BTrk.Pos4_Entry_TO_Pos4_Exit,
                  Item := "BTrk".A0301."B"["BTRK_A0301_Pos5.2_Long_PosAttesa"],
                  ENO => #_w5);
   "BTrk_Absence"(EN := #_w5, Item := "BTrk".A0301."B"["BTRK_A0301_Pos5.2_Long_Work_Pos"], ENO => #_w6);
   "BTrk_Absence"(EN := #_w6, Item := "BTrk".A0302_ENTRY."B"["BTRK_A0302_SPINTORE"], ENO => #_w7);
   #Ctrl.TRK.BTrk.Pos4_Entry_TO_Pos4_Exit := #_w7;
   #Ctrl.TRK.BTrk.Pos4_Entry_Cndz_To_Exit := #Ctrl.TRK.BTrk.Pos4_Entry_TO_Pos4_Exit AND #CIn.SpintoreLong.Ax_Sts.PosAttesa_Reached AND #CIn.P5.Spintore_Lat.Spin_Lat1.Rest AND #CIn.P5.Spintore_Lat.Spin_Lat2.Rest AND #CIn.P5.Sollevatori.Rest AND #Sts.P4.Fermi.Sens_Ing AND NOT #CIn.P5.SensUscitaBanco;
   #Ctrl.TRK.BTrk.Pos4_Entry_TO_Pos4_Exit := #Ctrl.TRK.BTrk.Pos4_Entry_Cndz_To_Exit AND #Sts.P4.Fermi.Sens_Out AND #CIn.P4.Fermi.Rest;
   IF #Ctrl.TRK.BTrk.Pos4_Entry_TO_Pos4_Exit THEN
       "BTrk".A0301."B"["BTRK_A0301_Pos4_Exit"] := "BTrk".A0301."B"["BTRK_A0301_Pos4_Entry"];
   END_IF;
   "BTrk_Presence"(EN := #Ctrl.TRK.BTrk.Pos4_Entry_TO_Pos4_Exit,
                   Item := "BTrk".A0301."B"["BTRK_A0301_Pos4_Exit"],
                   ENO => #_w8);
   IF #_w8 THEN "BTrk".A0301."B"["BTRK_A0301_Pos4_Entry"] := "BTrk".Empty; END_IF;
END_REGION

REGION Network 85: [P5] Movimento BTRK da Pos.4 Exit ==a==> Pos4_to_Pos5
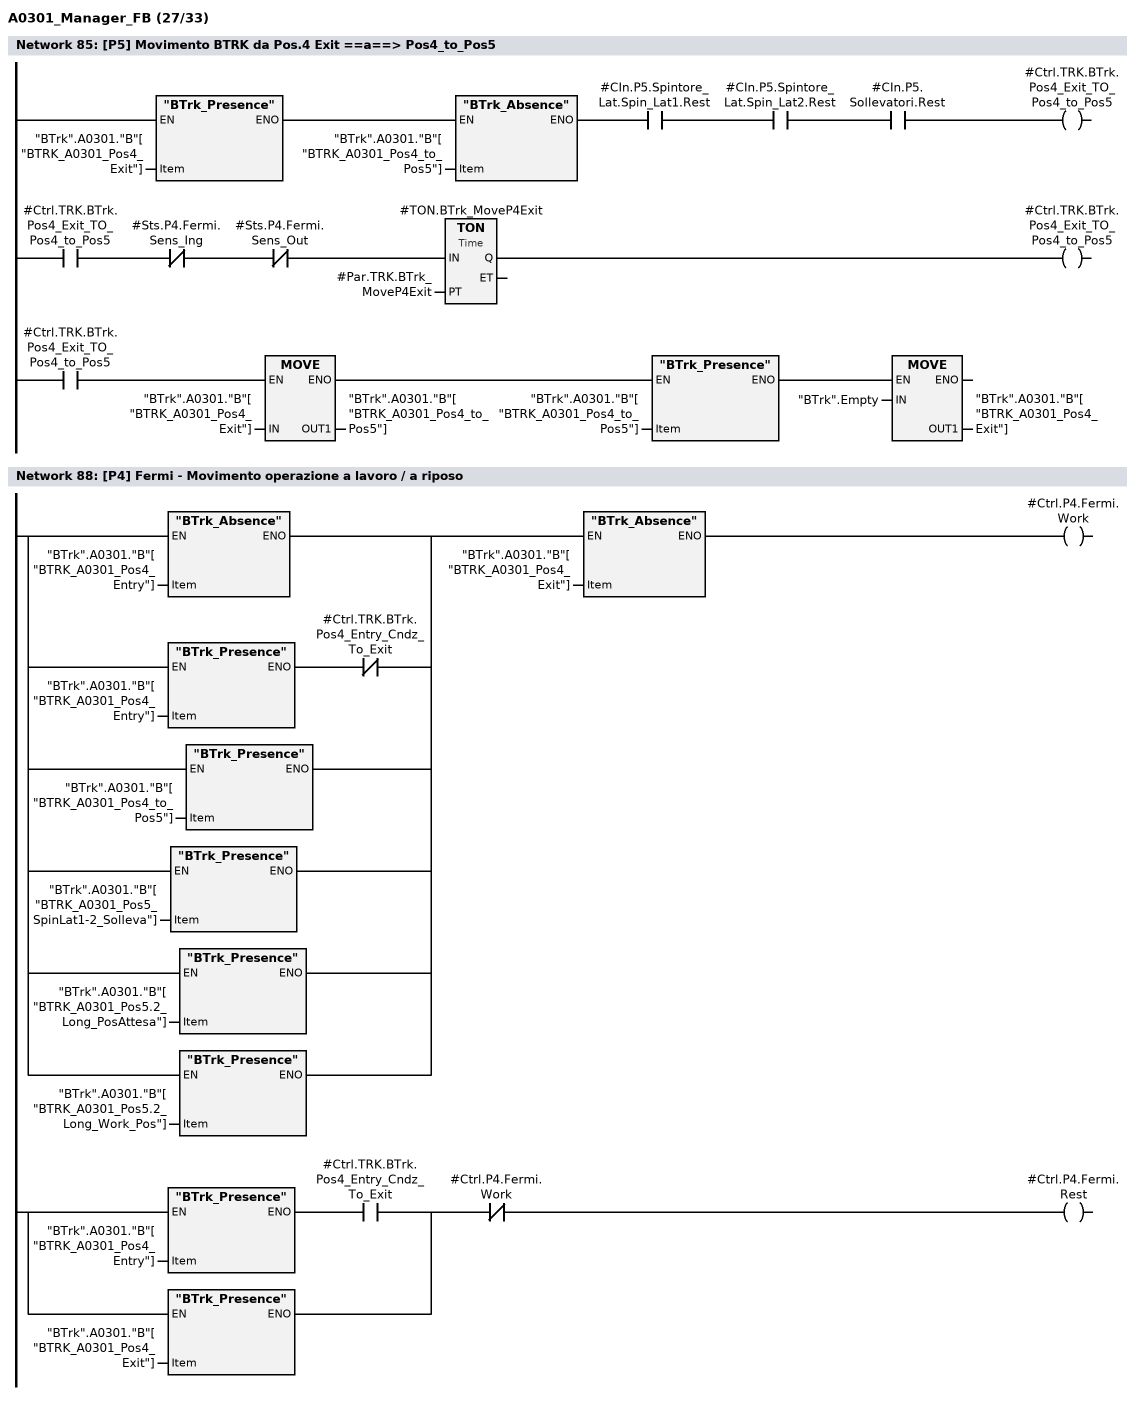
   RUNG wire#powerrail
      "BTrk_Presence"(Item := "BTrk".A0301."B"["BTRK_A0301_Pos4_Exit"])
      "BTrk_Absence"(Item := "BTrk".A0301."B"["BTRK_A0301_Pos4_to_Pos5"])
      Contact( #CIn.P5.Spintore_Lat.Spin_Lat1.Rest )
      Contact( #CIn.P5.Spintore_Lat.Spin_Lat2.Rest )
      Contact( #CIn.P5.Sollevatori.Rest )
      Coil( #Ctrl.TRK.BTrk.Pos4_Exit_TO_Pos4_to_Pos5 )
   END_RUNG
   RUNG wire#powerrail
      Contact( #Ctrl.TRK.BTrk.Pos4_Exit_TO_Pos4_to_Pos5 )
      I_Contact( #Sts.P4.Fermi.Sens_Ing )
      I_Contact( #Sts.P4.Fermi.Sens_Out )
      { S7_Templates := "time_type := Time" } #TON.BTrk_MoveP4Exit.TON(pt := #Par.TRK.BTrk_MoveP4Exit, et =>)
      Coil( #Ctrl.TRK.BTrk.Pos4_Exit_TO_Pos4_to_Pos5 )
   END_RUNG
   RUNG wire#powerrail
      Contact( #Ctrl.TRK.BTrk.Pos4_Exit_TO_Pos4_to_Pos5 )
      Move(in := "BTrk".A0301."B"["BTRK_A0301_Pos4_Exit"], out1 => "BTrk".A0301."B"["BTRK_A0301_Pos4_to_Pos5"])
      "BTrk_Presence"(Item := "BTrk".A0301."B"["BTRK_A0301_Pos4_to_Pos5"])
      Move(in := "BTrk".Empty, out1 => "BTrk".A0301."B"["BTRK_A0301_Pos4_Exit"])
   END_RUNG
   // the same network as SCL:
   "BTrk_Presence"(Item := "BTrk".A0301."B"["BTRK_A0301_Pos4_Exit"], ENO => #_w1);
   "BTrk_Absence"(EN := #_w1, Item := "BTrk".A0301."B"["BTRK_A0301_Pos4_to_Pos5"], ENO => #_w2);
   #Ctrl.TRK.BTrk.Pos4_Exit_TO_Pos4_to_Pos5 := #_w2 AND #CIn.P5.Spintore_Lat.Spin_Lat1.Rest AND #CIn.P5.Spintore_Lat.Spin_Lat2.Rest AND #CIn.P5.Sollevatori.Rest;
   #TON.BTrk_MoveP4Exit.TON(IN := #Ctrl.TRK.BTrk.Pos4_Exit_TO_Pos4_to_Pos5 AND NOT #Sts.P4.Fermi.Sens_Ing AND NOT #Sts.P4.Fermi.Sens_Out,
                           PT := #Par.TRK.BTrk_MoveP4Exit);
   #Ctrl.TRK.BTrk.Pos4_Exit_TO_Pos4_to_Pos5 := #TON.BTrk_MoveP4Exit.Q;
   IF #Ctrl.TRK.BTrk.Pos4_Exit_TO_Pos4_to_Pos5 THEN
       "BTrk".A0301."B"["BTRK_A0301_Pos4_to_Pos5"] := "BTrk".A0301."B"["BTRK_A0301_Pos4_Exit"];
   END_IF;
   "BTrk_Presence"(EN := #Ctrl.TRK.BTrk.Pos4_Exit_TO_Pos4_to_Pos5,
                   Item := "BTrk".A0301."B"["BTRK_A0301_Pos4_to_Pos5"],
                   ENO => #_w3);
   IF #_w3 THEN "BTrk".A0301."B"["BTRK_A0301_Pos4_Exit"] := "BTrk".Empty; END_IF;
END_REGION

REGION Network 87: [P4] <<< GESTIONE MOVIMENTO FERMI >>
END_REGION

REGION Network 88: [P4] Fermi - Movimento operazione a lavoro / a riposo
   RUNG wire#powerrail
      "BTrk_Absence"(Item := "BTrk".A0301."B"["BTRK_A0301_Pos4_Entry"])
      wire#w1
      "BTrk_Absence"(Item := "BTrk".A0301."B"["BTRK_A0301_Pos4_Exit"])
      Coil( #Ctrl.P4.Fermi.Work )
   END_RUNG
   RUNG wire#powerrail
      "BTrk_Presence"(Item := "BTrk".A0301."B"["BTRK_A0301_Pos4_Entry"])
      I_Contact( #Ctrl.TRK.BTrk.Pos4_Entry_Cndz_To_Exit )
   END_RUNG wire#w1
   RUNG wire#powerrail
      "BTrk_Presence"(Item := "BTrk".A0301."B"["BTRK_A0301_Pos4_to_Pos5"])
   END_RUNG wire#w1
   RUNG wire#powerrail
      "BTrk_Presence"(Item := "BTrk".A0301."B"["BTRK_A0301_Pos5_SpinLat1-2_Solleva"])
   END_RUNG wire#w1
   RUNG wire#powerrail
      "BTrk_Presence"(Item := "BTrk".A0301."B"["BTRK_A0301_Pos5.2_Long_PosAttesa"])
   END_RUNG wire#w1
   RUNG wire#powerrail
      "BTrk_Presence"(Item := "BTrk".A0301."B"["BTRK_A0301_Pos5.2_Long_Work_Pos"])
   END_RUNG wire#w1
   RUNG wire#powerrail
      "BTrk_Presence"(Item := "BTrk".A0301."B"["BTRK_A0301_Pos4_Entry"])
      Contact( #Ctrl.TRK.BTrk.Pos4_Entry_Cndz_To_Exit )
      wire#w2
      I_Contact( #Ctrl.P4.Fermi.Work )
      Coil( #Ctrl.P4.Fermi.Rest )
   END_RUNG
   RUNG wire#powerrail
      "BTrk_Presence"(Item := "BTrk".A0301."B"["BTRK_A0301_Pos4_Exit"])
   END_RUNG wire#w2
   // the same network as SCL:
   "BTrk_Absence"(Item := "BTrk".A0301."B"["BTRK_A0301_Pos4_Entry"], ENO => #_w1);
   "BTrk_Presence"(Item := "BTrk".A0301."B"["BTRK_A0301_Pos4_Entry"], ENO => #_w2);
   "BTrk_Presence"(Item := "BTrk".A0301."B"["BTRK_A0301_Pos4_to_Pos5"], ENO => #_w3);
   "BTrk_Presence"(Item := "BTrk".A0301."B"["BTRK_A0301_Pos5_SpinLat1-2_Solleva"], ENO => #_w4);
   "BTrk_Presence"(Item := "BTrk".A0301."B"["BTRK_A0301_Pos5.2_Long_PosAttesa"], ENO => #_w5);
   "BTrk_Presence"(Item := "BTrk".A0301."B"["BTRK_A0301_Pos5.2_Long_Work_Pos"], ENO => #_w6);
   "BTrk_Absence"(EN := #_w1 OR (#_w2 AND NOT #Ctrl.TRK.BTrk.Pos4_Entry_Cndz_To_Exit) OR #_w3 OR #_w4 OR #_w5 OR #_w6,
                  Item := "BTrk".A0301."B"["BTRK_A0301_Pos4_Exit"],
                  ENO => #_w7);
   #Ctrl.P4.Fermi.Work := #_w7;
   "BTrk_Presence"(Item := "BTrk".A0301."B"["BTRK_A0301_Pos4_Entry"], ENO => #_w8);
   "BTrk_Presence"(Item := "BTrk".A0301."B"["BTRK_A0301_Pos4_Exit"], ENO => #_w9);
   #Ctrl.P4.Fermi.Rest := ((#_w8 AND #Ctrl.TRK.BTrk.Pos4_Entry_Cndz_To_Exit) OR #_w9) AND NOT #Ctrl.P4.Fermi.Work;
END_REGION

REGION Network 89: [P4] Fermi - COut Manager
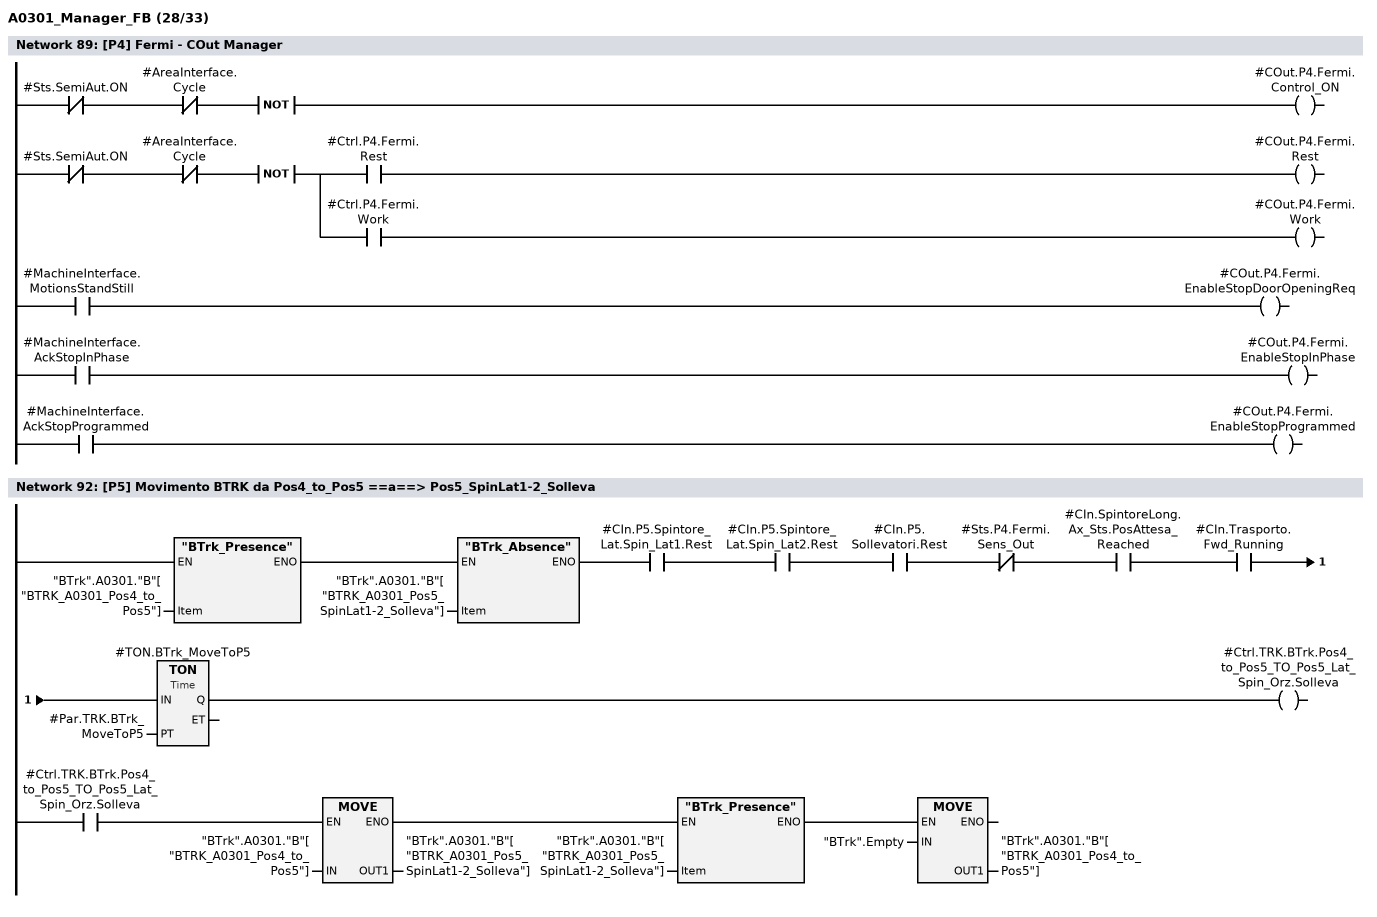
   RUNG wire#powerrail
      I_Contact( #Sts.SemiAut.ON )
      I_Contact( #AreaInterface.Cycle )
      Not()
      Coil( #COut.P4.Fermi.Control_ON )
   END_RUNG
   RUNG wire#powerrail
      I_Contact( #Sts.SemiAut.ON )
      I_Contact( #AreaInterface.Cycle )
      Not()
      wire#w1
      Contact( #Ctrl.P4.Fermi.Rest )
      Coil( #COut.P4.Fermi.Rest )
   END_RUNG
   RUNG wire#w1
      Contact( #Ctrl.P4.Fermi.Work )
      Coil( #COut.P4.Fermi.Work )
   END_RUNG
   RUNG wire#powerrail
      Contact( #MachineInterface.MotionsStandStill )
      Coil( #COut.P4.Fermi.EnableStopDoorOpeningReq )
   END_RUNG
   RUNG wire#powerrail
      Contact( #MachineInterface.AckStopInPhase )
      Coil( #COut.P4.Fermi.EnableStopInPhase )
   END_RUNG
   RUNG wire#powerrail
      Contact( #MachineInterface.AckStopProgrammed )
      Coil( #COut.P4.Fermi.EnableStopProgrammed )
   END_RUNG
   // the same network as SCL:
   #COut.P4.Fermi.Control_ON := NOT (NOT #Sts.SemiAut.ON AND NOT #AreaInterface.Cycle);
   #_w1 := NOT (NOT #Sts.SemiAut.ON AND NOT #AreaInterface.Cycle);
   #COut.P4.Fermi.Rest := #_w1 AND #Ctrl.P4.Fermi.Rest;
   #COut.P4.Fermi.Work := #_w1 AND #Ctrl.P4.Fermi.Work;
   #COut.P4.Fermi.EnableStopDoorOpeningReq := #MachineInterface.MotionsStandStill;
   #COut.P4.Fermi.EnableStopInPhase := #MachineInterface.AckStopInPhase;
   #COut.P4.Fermi.EnableStopProgrammed := #MachineInterface.AckStopProgrammed;
END_REGION

REGION Network 91: <<<<<<<<<<< POSIZIONE 5 >>>>>>>>>>>
END_REGION

REGION Network 92: [P5] Movimento BTRK da Pos4_to_Pos5 ==a==> Pos5_SpinLat1-2_Solleva
   RUNG wire#powerrail
      "BTrk_Presence"(Item := "BTrk".A0301."B"["BTRK_A0301_Pos4_to_Pos5"])
      "BTrk_Absence"(Item := "BTrk".A0301."B"["BTRK_A0301_Pos5_SpinLat1-2_Solleva"])
      Contact( #CIn.P5.Spintore_Lat.Spin_Lat1.Rest )
      Contact( #CIn.P5.Spintore_Lat.Spin_Lat2.Rest )
      Contact( #CIn.P5.Sollevatori.Rest )
      I_Contact( #Sts.P4.Fermi.Sens_Out )
      Contact( #CIn.SpintoreLong.Ax_Sts.PosAttesa_Reached )
      Contact( #CIn.Trasporto.Fwd_Running )
      { S7_Templates := "time_type := Time" } #TON.BTrk_MoveToP5.TON(pt := #Par.TRK.BTrk_MoveToP5, et =>)
      Coil( #Ctrl.TRK.BTrk.Pos4_to_Pos5_TO_Pos5_Lat_Spin_Orz.Solleva )
   END_RUNG
   RUNG wire#powerrail
      Contact( #Ctrl.TRK.BTrk.Pos4_to_Pos5_TO_Pos5_Lat_Spin_Orz.Solleva )
      Move(in := "BTrk".A0301."B"["BTRK_A0301_Pos4_to_Pos5"], out1 => "BTrk".A0301."B"["BTRK_A0301_Pos5_SpinLat1-2_Solleva"])
      "BTrk_Presence"(Item := "BTrk".A0301."B"["BTRK_A0301_Pos5_SpinLat1-2_Solleva"])
      Move(in := "BTrk".Empty, out1 => "BTrk".A0301."B"["BTRK_A0301_Pos4_to_Pos5"])
   END_RUNG
   // the same network as SCL:
   "BTrk_Presence"(Item := "BTrk".A0301."B"["BTRK_A0301_Pos4_to_Pos5"], ENO => #_w1);
   "BTrk_Absence"(EN := #_w1, Item := "BTrk".A0301."B"["BTRK_A0301_Pos5_SpinLat1-2_Solleva"], ENO => #_w2);
   #TON.BTrk_MoveToP5.TON(IN := #_w2 AND #CIn.P5.Spintore_Lat.Spin_Lat1.Rest AND #CIn.P5.Spintore_Lat.Spin_Lat2.Rest AND #CIn.P5.Sollevatori.Rest AND NOT #Sts.P4.Fermi.Sens_Out AND #CIn.SpintoreLong.Ax_Sts.PosAttesa_Reached AND #CIn.Trasporto.Fwd_Running,
                          PT := #Par.TRK.BTrk_MoveToP5);
   #Ctrl.TRK.BTrk.Pos4_to_Pos5_TO_Pos5_Lat_Spin_Orz.Solleva := #TON.BTrk_MoveToP5.Q;
   IF #Ctrl.TRK.BTrk.Pos4_to_Pos5_TO_Pos5_Lat_Spin_Orz.Solleva THEN
       "BTrk".A0301."B"["BTRK_A0301_Pos5_SpinLat1-2_Solleva"] := "BTrk".A0301."B"["BTRK_A0301_Pos4_to_Pos5"];
   END_IF;
   "BTrk_Presence"(EN := #Ctrl.TRK.BTrk.Pos4_to_Pos5_TO_Pos5_Lat_Spin_Orz.Solleva,
                   Item := "BTrk".A0301."B"["BTRK_A0301_Pos5_SpinLat1-2_Solleva"],
                   ENO => #_w3);
   IF #_w3 THEN "BTrk".A0301."B"["BTRK_A0301_Pos4_to_Pos5"] := "BTrk".Empty; END_IF;
END_REGION

REGION Network 94: [P5] <<< GESTIONE MOVIMENTO SPINTORI LATERALI - SOLLEVATORI >>>
END_REGION

REGION Network 95: [P5] Spintore Laterale - Movimento operazione a lavoro / a riposo
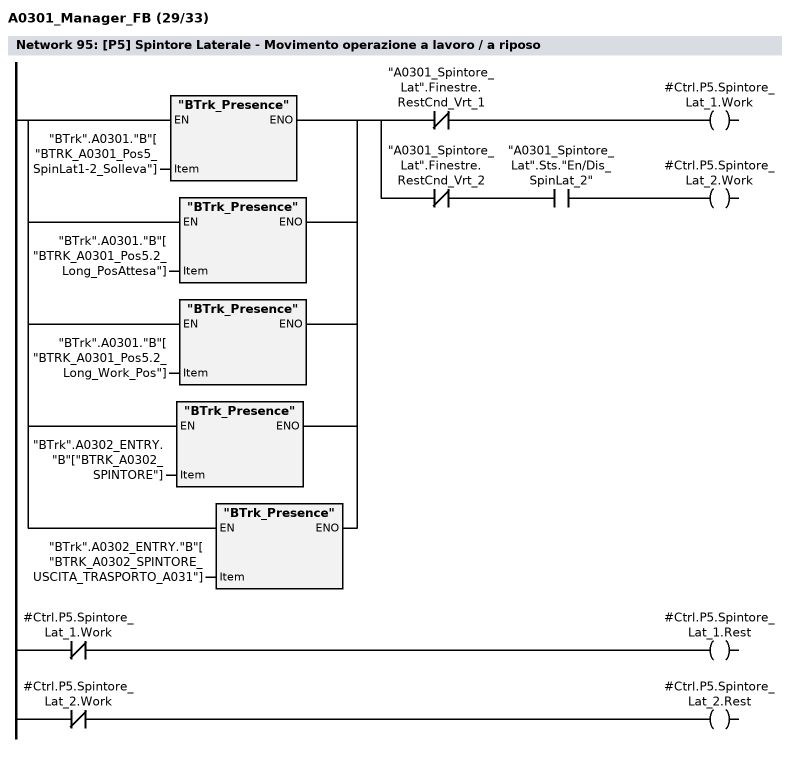
   RUNG wire#powerrail
      "BTrk_Presence"(Item := "BTrk".A0301."B"["BTRK_A0301_Pos5_SpinLat1-2_Solleva"])
      wire#w1
      I_Contact( "A0301_Spintore_Lat".Finestre.RestCnd_Vrt_1 )
      Coil( #Ctrl.P5.Spintore_Lat_1.Work )
   END_RUNG
   RUNG wire#powerrail
      "BTrk_Presence"(Item := "BTrk".A0301."B"["BTRK_A0301_Pos5.2_Long_PosAttesa"])
   END_RUNG wire#w1
   RUNG wire#powerrail
      "BTrk_Presence"(Item := "BTrk".A0301."B"["BTRK_A0301_Pos5.2_Long_Work_Pos"])
   END_RUNG wire#w1
   RUNG wire#powerrail
      "BTrk_Presence"(Item := "BTrk".A0302_ENTRY."B"["BTRK_A0302_SPINTORE"])
   END_RUNG wire#w1
   RUNG wire#powerrail
      "BTrk_Presence"(Item := "BTrk".A0302_ENTRY."B"["BTRK_A0302_SPINTORE_USCITA_TRASPORTO_A031"])
   END_RUNG wire#w1
   RUNG wire#w1
      I_Contact( "A0301_Spintore_Lat".Finestre.RestCnd_Vrt_2 )
      Contact( "A0301_Spintore_Lat".Sts."En/Dis_SpinLat_2" )
      Coil( #Ctrl.P5.Spintore_Lat_2.Work )
   END_RUNG
   RUNG wire#powerrail
      I_Contact( #Ctrl.P5.Spintore_Lat_1.Work )
      Coil( #Ctrl.P5.Spintore_Lat_1.Rest )
   END_RUNG
   RUNG wire#powerrail
      I_Contact( #Ctrl.P5.Spintore_Lat_2.Work )
      Coil( #Ctrl.P5.Spintore_Lat_2.Rest )
   END_RUNG
   // the same network as SCL:
   "BTrk_Presence"(Item := "BTrk".A0301."B"["BTRK_A0301_Pos5_SpinLat1-2_Solleva"], ENO => #_w1);
   "BTrk_Presence"(Item := "BTrk".A0301."B"["BTRK_A0301_Pos5.2_Long_PosAttesa"], ENO => #_w2);
   "BTrk_Presence"(Item := "BTrk".A0301."B"["BTRK_A0301_Pos5.2_Long_Work_Pos"], ENO => #_w3);
   "BTrk_Presence"(Item := "BTrk".A0302_ENTRY."B"["BTRK_A0302_SPINTORE"], ENO => #_w4);
   "BTrk_Presence"(Item := "BTrk".A0302_ENTRY."B"["BTRK_A0302_SPINTORE_USCITA_TRASPORTO_A031"], ENO => #_w5);
   #_w6 := #_w1 OR #_w2 OR #_w3 OR #_w4 OR #_w5;
   #Ctrl.P5.Spintore_Lat_1.Work := #_w6 AND NOT "A0301_Spintore_Lat".Finestre.RestCnd_Vrt_1;
   #Ctrl.P5.Spintore_Lat_2.Work := #_w6 AND NOT "A0301_Spintore_Lat".Finestre.RestCnd_Vrt_2 AND "A0301_Spintore_Lat".Sts."En/Dis_SpinLat_2";
   #Ctrl.P5.Spintore_Lat_1.Rest := NOT #Ctrl.P5.Spintore_Lat_1.Work;
   #Ctrl.P5.Spintore_Lat_2.Rest := NOT #Ctrl.P5.Spintore_Lat_2.Work;
END_REGION

REGION Network 96: [P5] Spintore Laterale - COut Manager
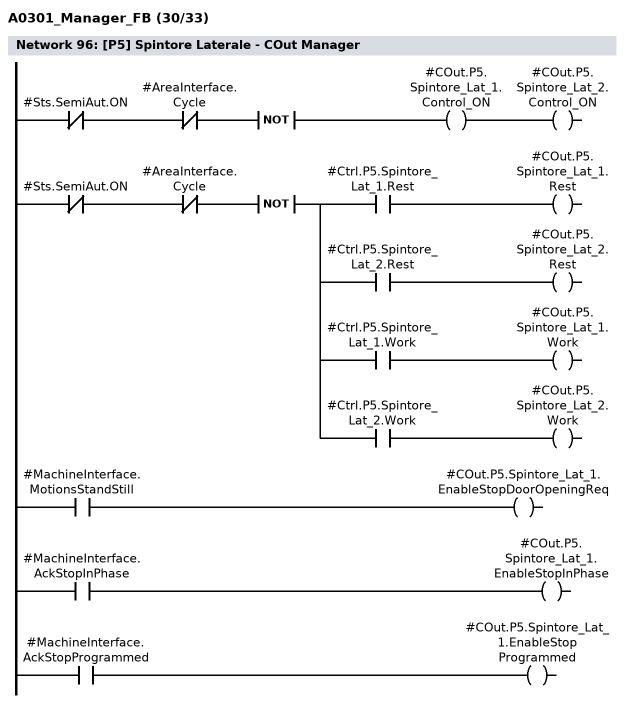
   RUNG wire#powerrail
      I_Contact( #Sts.SemiAut.ON )
      I_Contact( #AreaInterface.Cycle )
      Not()
      Coil( #COut.P5.Spintore_Lat_1.Control_ON )
      Coil( #COut.P5.Spintore_Lat_2.Control_ON )
   END_RUNG
   RUNG wire#powerrail
      I_Contact( #Sts.SemiAut.ON )
      I_Contact( #AreaInterface.Cycle )
      Not()
      wire#w1
      Contact( #Ctrl.P5.Spintore_Lat_1.Rest )
      Coil( #COut.P5.Spintore_Lat_1.Rest )
   END_RUNG
   RUNG wire#w1
      Contact( #Ctrl.P5.Spintore_Lat_2.Rest )
      Coil( #COut.P5.Spintore_Lat_2.Rest )
   END_RUNG
   RUNG wire#w1
      Contact( #Ctrl.P5.Spintore_Lat_1.Work )
      Coil( #COut.P5.Spintore_Lat_1.Work )
   END_RUNG
   RUNG wire#w1
      Contact( #Ctrl.P5.Spintore_Lat_2.Work )
      Coil( #COut.P5.Spintore_Lat_2.Work )
   END_RUNG
   RUNG wire#powerrail
      Contact( #MachineInterface.MotionsStandStill )
      Coil( #COut.P5.Spintore_Lat_1.EnableStopDoorOpeningReq )
   END_RUNG
   RUNG wire#powerrail
      Contact( #MachineInterface.AckStopInPhase )
      Coil( #COut.P5.Spintore_Lat_1.EnableStopInPhase )
   END_RUNG
   RUNG wire#powerrail
      Contact( #MachineInterface.AckStopProgrammed )
      Coil( #COut.P5.Spintore_Lat_1.EnableStopProgrammed )
   END_RUNG
   // the same network as SCL:
   #COut.P5.Spintore_Lat_1.Control_ON := NOT (NOT #Sts.SemiAut.ON AND NOT #AreaInterface.Cycle);
   #COut.P5.Spintore_Lat_2.Control_ON := #COut.P5.Spintore_Lat_1.Control_ON;
   #_w1 := NOT (NOT #Sts.SemiAut.ON AND NOT #AreaInterface.Cycle);
   #COut.P5.Spintore_Lat_1.Rest := #_w1 AND #Ctrl.P5.Spintore_Lat_1.Rest;
   #COut.P5.Spintore_Lat_2.Rest := #_w1 AND #Ctrl.P5.Spintore_Lat_2.Rest;
   #COut.P5.Spintore_Lat_1.Work := #_w1 AND #Ctrl.P5.Spintore_Lat_1.Work;
   #COut.P5.Spintore_Lat_2.Work := #_w1 AND #Ctrl.P5.Spintore_Lat_2.Work;
   #COut.P5.Spintore_Lat_1.EnableStopDoorOpeningReq := #MachineInterface.MotionsStandStill;
   #COut.P5.Spintore_Lat_1.EnableStopInPhase := #MachineInterface.AckStopInPhase;
   #COut.P5.Spintore_Lat_1.EnableStopProgrammed := #MachineInterface.AckStopProgrammed;
END_REGION

REGION Network 97: [P5] Sollevatori - Movimento operazione a lavoro / a riposo
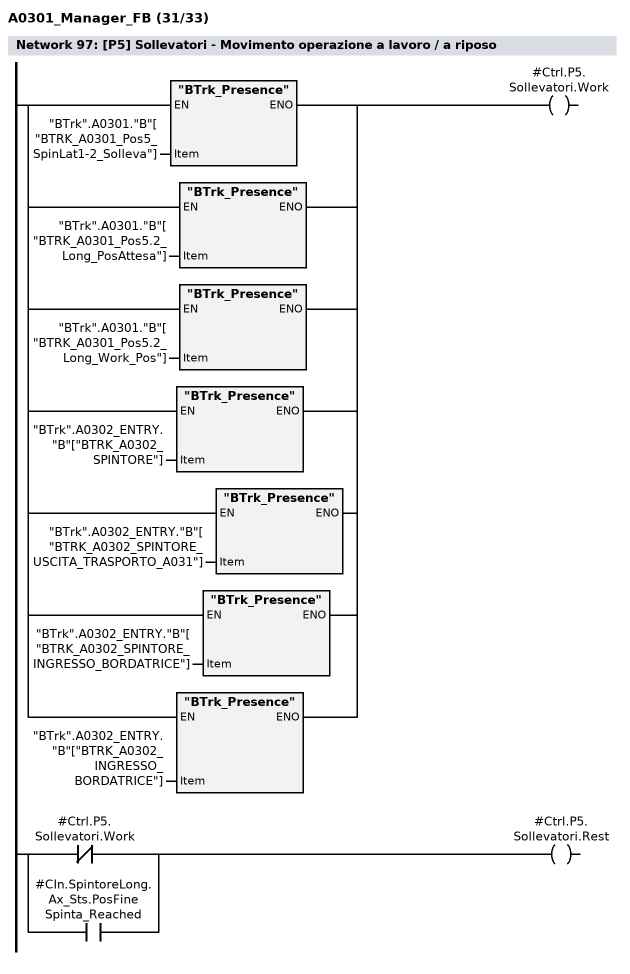
   RUNG wire#powerrail
      "BTrk_Presence"(Item := "BTrk".A0301."B"["BTRK_A0301_Pos5_SpinLat1-2_Solleva"])
      wire#w1
      Coil( #Ctrl.P5.Sollevatori.Work )
   END_RUNG
   RUNG wire#powerrail
      "BTrk_Presence"(Item := "BTrk".A0301."B"["BTRK_A0301_Pos5.2_Long_PosAttesa"])
   END_RUNG wire#w1
   RUNG wire#powerrail
      "BTrk_Presence"(Item := "BTrk".A0301."B"["BTRK_A0301_Pos5.2_Long_Work_Pos"])
   END_RUNG wire#w1
   RUNG wire#powerrail
      "BTrk_Presence"(Item := "BTrk".A0302_ENTRY."B"["BTRK_A0302_SPINTORE"])
   END_RUNG wire#w1
   RUNG wire#powerrail
      "BTrk_Presence"(Item := "BTrk".A0302_ENTRY."B"["BTRK_A0302_SPINTORE_USCITA_TRASPORTO_A031"])
   END_RUNG wire#w1
   RUNG wire#powerrail
      "BTrk_Presence"(Item := "BTrk".A0302_ENTRY."B"["BTRK_A0302_SPINTORE_INGRESSO_BORDATRICE"])
   END_RUNG wire#w1
   RUNG wire#powerrail
      "BTrk_Presence"(Item := "BTrk".A0302_ENTRY."B"["BTRK_A0302_INGRESSO_BORDATRICE"])
   END_RUNG wire#w1
   RUNG wire#powerrail
      I_Contact( #Ctrl.P5.Sollevatori.Work )
      wire#w2
      Coil( #Ctrl.P5.Sollevatori.Rest )
   END_RUNG
   RUNG wire#powerrail
      Contact( #CIn.SpintoreLong.Ax_Sts.PosFineSpinta_Reached )
   END_RUNG wire#w2
   // the same network as SCL:
   "BTrk_Presence"(Item := "BTrk".A0301."B"["BTRK_A0301_Pos5_SpinLat1-2_Solleva"], ENO => #_w1);
   "BTrk_Presence"(Item := "BTrk".A0301."B"["BTRK_A0301_Pos5.2_Long_PosAttesa"], ENO => #_w2);
   "BTrk_Presence"(Item := "BTrk".A0301."B"["BTRK_A0301_Pos5.2_Long_Work_Pos"], ENO => #_w3);
   "BTrk_Presence"(Item := "BTrk".A0302_ENTRY."B"["BTRK_A0302_SPINTORE"], ENO => #_w4);
   "BTrk_Presence"(Item := "BTrk".A0302_ENTRY."B"["BTRK_A0302_SPINTORE_USCITA_TRASPORTO_A031"], ENO => #_w5);
   "BTrk_Presence"(Item := "BTrk".A0302_ENTRY."B"["BTRK_A0302_SPINTORE_INGRESSO_BORDATRICE"], ENO => #_w6);
   "BTrk_Presence"(Item := "BTrk".A0302_ENTRY."B"["BTRK_A0302_INGRESSO_BORDATRICE"], ENO => #_w7);
   #Ctrl.P5.Sollevatori.Work := #_w1 OR #_w2 OR #_w3 OR #_w4 OR #_w5 OR #_w6 OR #_w7;
   #Ctrl.P5.Sollevatori.Rest := NOT #Ctrl.P5.Sollevatori.Work OR #CIn.SpintoreLong.Ax_Sts.PosFineSpinta_Reached;
END_REGION

REGION Network 98: [P5] Sollevatori - COut Manager
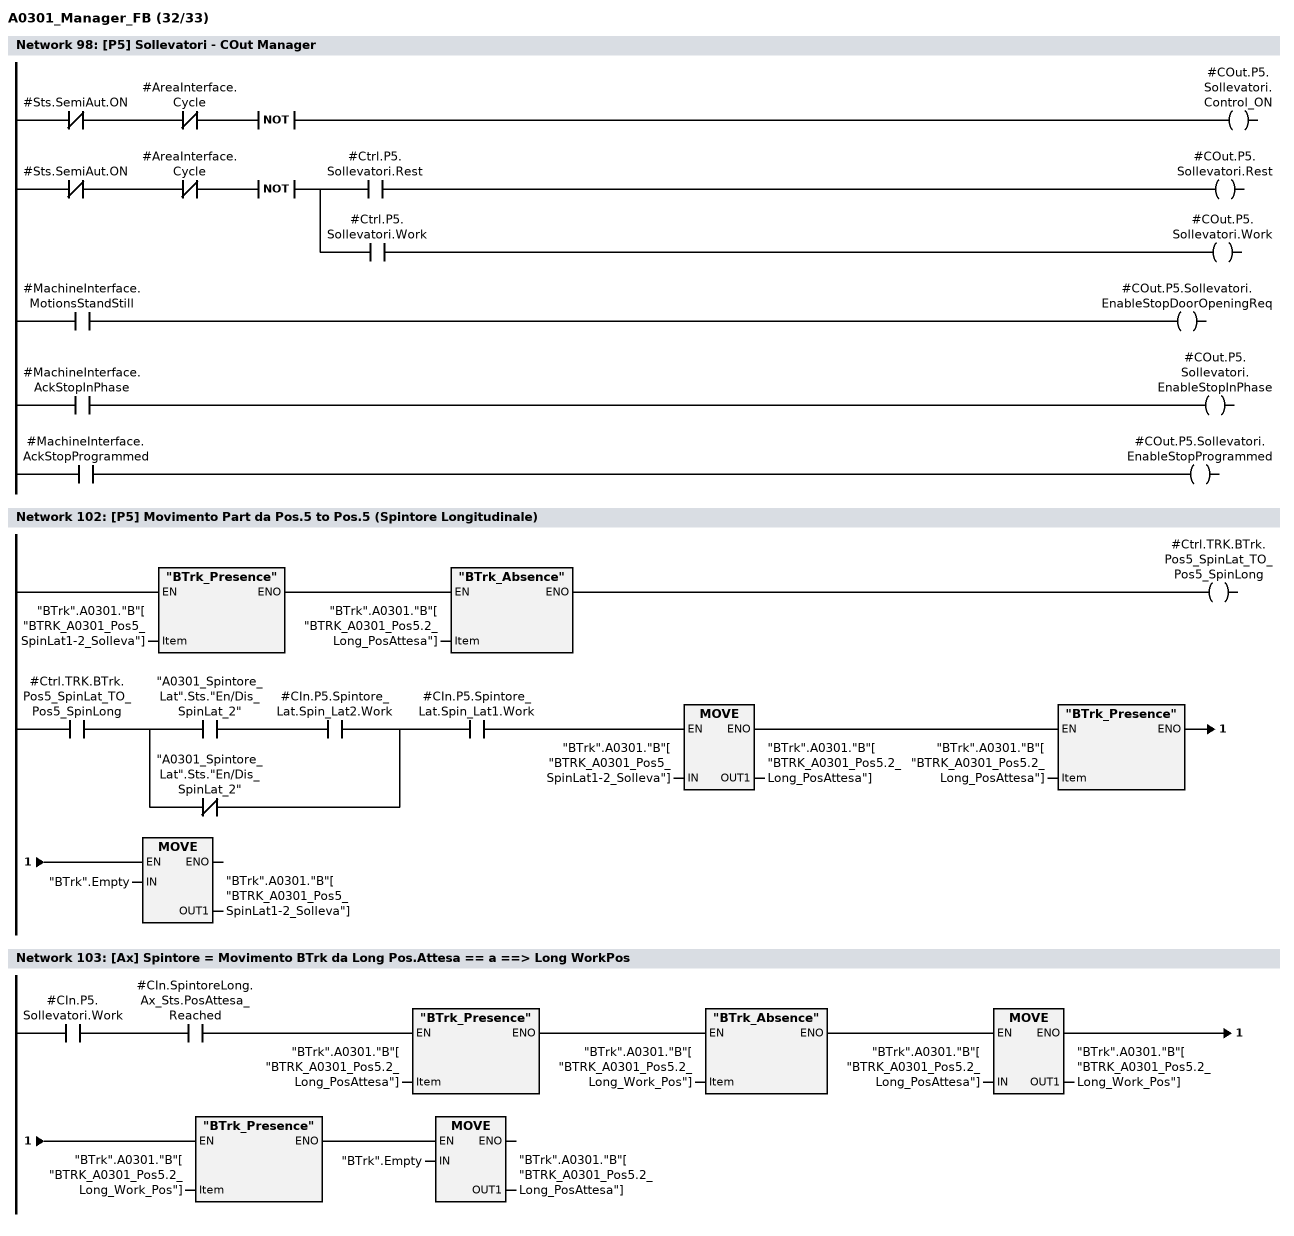
   RUNG wire#powerrail
      I_Contact( #Sts.SemiAut.ON )
      I_Contact( #AreaInterface.Cycle )
      Not()
      Coil( #COut.P5.Sollevatori.Control_ON )
   END_RUNG
   RUNG wire#powerrail
      I_Contact( #Sts.SemiAut.ON )
      I_Contact( #AreaInterface.Cycle )
      Not()
      wire#w1
      Contact( #Ctrl.P5.Sollevatori.Rest )
      Coil( #COut.P5.Sollevatori.Rest )
   END_RUNG
   RUNG wire#w1
      Contact( #Ctrl.P5.Sollevatori.Work )
      Coil( #COut.P5.Sollevatori.Work )
   END_RUNG
   RUNG wire#powerrail
      Contact( #MachineInterface.MotionsStandStill )
      Coil( #COut.P5.Sollevatori.EnableStopDoorOpeningReq )
   END_RUNG
   RUNG wire#powerrail
      Contact( #MachineInterface.AckStopInPhase )
      Coil( #COut.P5.Sollevatori.EnableStopInPhase )
   END_RUNG
   RUNG wire#powerrail
      Contact( #MachineInterface.AckStopProgrammed )
      Coil( #COut.P5.Sollevatori.EnableStopProgrammed )
   END_RUNG
   // the same network as SCL:
   #COut.P5.Sollevatori.Control_ON := NOT (NOT #Sts.SemiAut.ON AND NOT #AreaInterface.Cycle);
   #_w1 := NOT (NOT #Sts.SemiAut.ON AND NOT #AreaInterface.Cycle);
   #COut.P5.Sollevatori.Rest := #_w1 AND #Ctrl.P5.Sollevatori.Rest;
   #COut.P5.Sollevatori.Work := #_w1 AND #Ctrl.P5.Sollevatori.Work;
   #COut.P5.Sollevatori.EnableStopDoorOpeningReq := #MachineInterface.MotionsStandStill;
   #COut.P5.Sollevatori.EnableStopInPhase := #MachineInterface.AckStopInPhase;
   #COut.P5.Sollevatori.EnableStopProgrammed := #MachineInterface.AckStopProgrammed;
END_REGION

REGION Network 100: [P5] <<< GESTIONE MOVIMENTO SPINTORE LONGITUDINALE >>
END_REGION

REGION Network 102: [P5] Movimento Part da Pos.5 to Pos.5 (Spintore Longitudinale)
   RUNG wire#powerrail
      "BTrk_Presence"(Item := "BTrk".A0301."B"["BTRK_A0301_Pos5_SpinLat1-2_Solleva"])
      "BTrk_Absence"(Item := "BTrk".A0301."B"["BTRK_A0301_Pos5.2_Long_PosAttesa"])
      Coil( #Ctrl.TRK.BTrk.Pos5_SpinLat_TO_Pos5_SpinLong )
   END_RUNG
   RUNG wire#powerrail
      Contact( #Ctrl.TRK.BTrk.Pos5_SpinLat_TO_Pos5_SpinLong )
      wire#w1
      Contact( "A0301_Spintore_Lat".Sts."En/Dis_SpinLat_2" )
      Contact( #CIn.P5.Spintore_Lat.Spin_Lat2.Work )
      wire#w2
      Contact( #CIn.P5.Spintore_Lat.Spin_Lat1.Work )
      Move(in := "BTrk".A0301."B"["BTRK_A0301_Pos5_SpinLat1-2_Solleva"], out1 => "BTrk".A0301."B"["BTRK_A0301_Pos5.2_Long_PosAttesa"])
      "BTrk_Presence"(Item := "BTrk".A0301."B"["BTRK_A0301_Pos5.2_Long_PosAttesa"])
      Move(in := "BTrk".Empty, out1 => "BTrk".A0301."B"["BTRK_A0301_Pos5_SpinLat1-2_Solleva"])
   END_RUNG
   RUNG wire#w1
      I_Contact( "A0301_Spintore_Lat".Sts."En/Dis_SpinLat_2" )
   END_RUNG wire#w2
   // the same network as SCL:
   "BTrk_Presence"(Item := "BTrk".A0301."B"["BTRK_A0301_Pos5_SpinLat1-2_Solleva"], ENO => #_w1);
   "BTrk_Absence"(EN := #_w1, Item := "BTrk".A0301."B"["BTRK_A0301_Pos5.2_Long_PosAttesa"], ENO => #_w2);
   #Ctrl.TRK.BTrk.Pos5_SpinLat_TO_Pos5_SpinLong := #_w2;
   IF #Ctrl.TRK.BTrk.Pos5_SpinLat_TO_Pos5_SpinLong AND (("A0301_Spintore_Lat".Sts."En/Dis_SpinLat_2" AND #CIn.P5.Spintore_Lat.Spin_Lat2.Work) OR NOT "A0301_Spintore_Lat".Sts."En/Dis_SpinLat_2") AND #CIn.P5.Spintore_Lat.Spin_Lat1.Work THEN
       "BTrk".A0301."B"["BTRK_A0301_Pos5.2_Long_PosAttesa"] := "BTrk".A0301."B"["BTRK_A0301_Pos5_SpinLat1-2_Solleva"];
   END_IF;
   "BTrk_Presence"(EN := #Ctrl.TRK.BTrk.Pos5_SpinLat_TO_Pos5_SpinLong AND (("A0301_Spintore_Lat".Sts."En/Dis_SpinLat_2" AND #CIn.P5.Spintore_Lat.Spin_Lat2.Work) OR NOT "A0301_Spintore_Lat".Sts."En/Dis_SpinLat_2") AND #CIn.P5.Spintore_Lat.Spin_Lat1.Work,
                   Item := "BTrk".A0301."B"["BTRK_A0301_Pos5.2_Long_PosAttesa"],
                   ENO => #_w3);
   IF #_w3 THEN "BTrk".A0301."B"["BTRK_A0301_Pos5_SpinLat1-2_Solleva"] := "BTrk".Empty; END_IF;
END_REGION

REGION Network 103: [Ax] Spintore = Movimento BTrk da Long Pos.Attesa == a ==> Long WorkPos
   RUNG wire#powerrail
      Contact( #CIn.P5.Sollevatori.Work )
      Contact( #CIn.SpintoreLong.Ax_Sts.PosAttesa_Reached )
      "BTrk_Presence"(Item := "BTrk".A0301."B"["BTRK_A0301_Pos5.2_Long_PosAttesa"])
      "BTrk_Absence"(Item := "BTrk".A0301."B"["BTRK_A0301_Pos5.2_Long_Work_Pos"])
      Move(in := "BTrk".A0301."B"["BTRK_A0301_Pos5.2_Long_PosAttesa"], out1 => "BTrk".A0301."B"["BTRK_A0301_Pos5.2_Long_Work_Pos"])
      "BTrk_Presence"(Item := "BTrk".A0301."B"["BTRK_A0301_Pos5.2_Long_Work_Pos"])
      Move(in := "BTrk".Empty, out1 => "BTrk".A0301."B"["BTRK_A0301_Pos5.2_Long_PosAttesa"])
   END_RUNG
   // the same network as SCL:
   "BTrk_Presence"(EN := #CIn.P5.Sollevatori.Work AND #CIn.SpintoreLong.Ax_Sts.PosAttesa_Reached,
                   Item := "BTrk".A0301."B"["BTRK_A0301_Pos5.2_Long_PosAttesa"],
                   ENO => #_w1);
   "BTrk_Absence"(EN := #_w1, Item := "BTrk".A0301."B"["BTRK_A0301_Pos5.2_Long_Work_Pos"], ENO => #_w2);
   IF #_w2 THEN
       "BTrk".A0301."B"["BTRK_A0301_Pos5.2_Long_Work_Pos"] := "BTrk".A0301."B"["BTRK_A0301_Pos5.2_Long_PosAttesa"];
   END_IF;
   "BTrk_Presence"(EN := #_w2, Item := "BTrk".A0301."B"["BTRK_A0301_Pos5.2_Long_Work_Pos"], ENO => #_w3);
   IF #_w3 THEN "BTrk".A0301."B"["BTRK_A0301_Pos5.2_Long_PosAttesa"] := "BTrk".Empty; END_IF;
END_REGION

REGION Network 104: [P5] <<< GESTIONE MOVIMENTO SPINTORE LONGITUDINALE >>
END_REGION

REGION Network 105: <+>
END_REGION

REGION Network 106: Stop Cycle
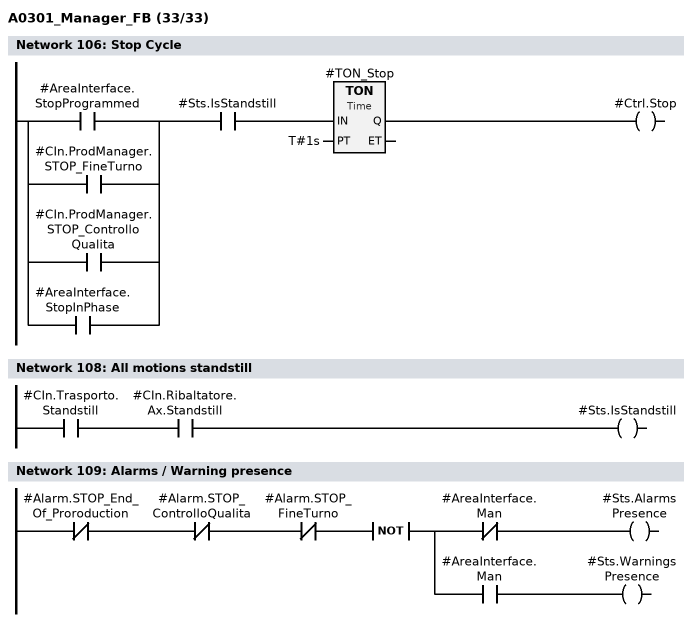
   RUNG wire#powerrail
      Contact( #AreaInterface.StopProgrammed )
      wire#w1
      Contact( #Sts.IsStandstill )
      { S7_Templates := "time_type := Time" } #TON_Stop.TON(pt := T#1s, et =>)
      Coil( #Ctrl.Stop )
   END_RUNG
   RUNG wire#powerrail
      Contact( #CIn.ProdManager.STOP_FineTurno )
   END_RUNG wire#w1
   RUNG wire#powerrail
      Contact( #CIn.ProdManager.STOP_ControlloQualita )
   END_RUNG wire#w1
   RUNG wire#powerrail
      Contact( #AreaInterface.StopInPhase )
   END_RUNG wire#w1
   // the same network as SCL:
   #TON_Stop.TON(IN := (#AreaInterface.StopProgrammed OR #CIn.ProdManager.STOP_FineTurno OR #CIn.ProdManager.STOP_ControlloQualita OR #AreaInterface.StopInPhase) AND #Sts.IsStandstill,
                 PT := T#1s);
   #Ctrl.Stop := #TON_Stop.Q;
END_REGION

REGION Network 107: << FINAL OPERATIONS >>
   // +
   // +
   // +
   // +
   // +
   // +
   // +
   // +
   // +
   // +
   // +
   // +
   // +
END_REGION

REGION Network 108: All motions standstill
   RUNG wire#powerrail
      Contact( #CIn.Trasporto.Standstill )
      Contact( #CIn.Ribaltatore.Ax.Standstill )
      Coil( #Sts.IsStandstill )
   END_RUNG
   // the same network as SCL:
   #Sts.IsStandstill := #CIn.Trasporto.Standstill AND #CIn.Ribaltatore.Ax.Standstill;
END_REGION

REGION Network 109: Alarms / Warning presence
   RUNG wire#powerrail
      I_Contact( #Alarm.STOP_End_Of_Proroduction )
      I_Contact( #Alarm.STOP_ControlloQualita )
      I_Contact( #Alarm.STOP_FineTurno )
      Not()
      wire#w1
      I_Contact( #AreaInterface.Man )
      Coil( #Sts.AlarmsPresence )
   END_RUNG
   RUNG wire#w1
      Contact( #AreaInterface.Man )
      Coil( #Sts.WarningsPresence )
   END_RUNG
   // the same network as SCL:
   #_w1 := NOT (NOT #Alarm.STOP_End_Of_Proroduction AND NOT #Alarm.STOP_ControlloQualita AND NOT #Alarm.STOP_FineTurno);
   #Sts.AlarmsPresence := #_w1 AND NOT #AreaInterface.Man;
   #Sts.WarningsPresence := #_w1 AND #AreaInterface.Man;
END_REGION

REGION Network 110 (SCL): Collect machine to area interface
   #MachineInterface.AlarmsPresence := #Sts.AlarmsPresence;

   #MachineInterface.WarningPresence := #Sts.WarningsPresence;

   #MachineInterface.MotionsStandStill := #Sts.IsStandstill;

   #MachineInterface.AutReady := #AreaInterface.Aut AND NOT #Sts.AlarmsPresence;


   #MachineInterface.AckStopInPhase := #AreaInterface.StopInPhase AND #Ctrl.Stop;

   #MachineInterface.AckStopProgrammed := #AreaInterface.StopProgrammed AND #Ctrl.Stop;


   #MachineInterface.Aborting := #AreaInterface.Aut AND #Sts.AlarmsPresence;
END_REGION
END_FUNCTION_BLOCK
